## Short summary
This assertion method checks if the current value is inside a limit

**Attention:** 
	limits are included: ``valueIsInRangeOf(ldt#1970-01-01-0:0:0, ldt#1970-01-01-0:0:0, ldt#1970-01-01-0:0:0)``
	is a true assertion

.. <legal notes>

legal notes
=================
| SPDX-FileCopyrightText: © 2022 ekvip automation GmbH <info@ekvip.de>
| SPDX-License-Identifier: Apache-2.0
| For details check: Apache-2.0_

.. _Apache-2.0: https://www.apache.org/licenses/LICENSE-2.0

.. </legal notes>



*)

METHOD valueIsInRangeOf
VAR_INPUT
	(* lower limit for the current value *)
	lowerLimit		:LDT;
	(* current value to check *)
	currentValue	:LDT;
	(* upper limit for the current value *)
	upperLimit		:LDT;
	(* message if the assertion is false *)
	message			:AssertMessage;
END_VAR
IF (
	(currentValue < lowerLimit)
	OR (currentValue > upperLimit)
) THEN
	THIS^.assertionWasWrong(message, THIS^.getDebugInfo('valueIsInRangeOf'));
END_IF
END_METHOD

(*

## Short summary
This assertion method checks if the current value is less than the greater value

.. <legal notes>

legal notes
=================
| SPDX-FileCopyrightText: © 2022 ekvip automation GmbH <info@ekvip.de>
| SPDX-License-Identifier: Apache-2.0
| For details check: Apache-2.0_

.. _Apache-2.0: https://www.apache.org/licenses/LICENSE-2.0

.. </legal notes>



*)

METHOD valueIsLessThan
VAR_INPUT
	(* current value to check *)
	currentValue	:LDT;
	(* greater than upper limit *)
	greaterValue	:LDT;
	(* message if the assertion is false *)
	message			:AssertMessage;
END_VAR
IF (currentValue >= greaterValue) THEN
	THIS^.assertionWasWrong(message, THIS^.getDebugInfo('valueIsLessThan'));
END_IF
END_METHOD

(*

## Short summary
This assertion method checks if the current value is less than or equal to the maximum value

.. <legal notes>

legal notes
=================
| SPDX-FileCopyrightText: © 2022 ekvip automation GmbH <info@ekvip.de>
| SPDX-License-Identifier: Apache-2.0
| For details check: Apache-2.0_

.. _Apache-2.0: https://www.apache.org/licenses/LICENSE-2.0

.. </legal notes>



*)

METHOD valueIsMax
VAR_INPUT
	(* current value to check *)
	currentValue	:LDT;
	(* upper limit for the current value *)
	maximumValue	:LDT;
	(* message if the assertion is false *)
	message			:AssertMessage;
END_VAR
IF (currentValue > maximumValue) THEN
	THIS^.assertionWasWrong(message, THIS^.getDebugInfo('valueIsMax'));
END_IF
END_METHOD

(*

## Short summary
This assertion method checks if the current value is greater than or equal to the minimum value

.. <legal notes>

legal notes
=================
| SPDX-FileCopyrightText: © 2022 ekvip automation GmbH <info@ekvip.de>
| SPDX-License-Identifier: Apache-2.0
| For details check: Apache-2.0_

.. _Apache-2.0: https://www.apache.org/licenses/LICENSE-2.0

.. </legal notes>



*)

METHOD valueIsMin
VAR_INPUT
	(* current value to check *)
	currentValue	:LDT;
	(* lower limit for the current value *)
	minimumValue	:LDT;
	(* message if the assertion is false *)
	message			:AssertMessage;
END_VAR
IF (currentValue < minimumValue) THEN
	THIS^.assertionWasWrong(message, THIS^.getDebugInfo('valueIsMin'));
END_IF
END_METHOD

(*

## Short summary
This assertion method checks if the current value is not equal to the unexpected value

.. <legal notes>

legal notes
=================
| SPDX-FileCopyrightText: © 2022 ekvip automation GmbH <info@ekvip.de>
| SPDX-License-Identifier: Apache-2.0
| For details check: Apache-2.0_

.. _Apache-2.0: https://www.apache.org/licenses/LICENSE-2.0

.. </legal notes>



*)

METHOD valueIsNotEqualTo
VAR_INPUT
	(* current value to check *)
	currentValue	:LDT;
	(* unexpected value to compare *)
	unexpectedValue	:LDT;
	(* message if the assertion is false *)
	message			:AssertMessage;
END_VAR
IF (currentValue = unexpectedValue) THEN
	THIS^.assertionWasWrong(message, THIS^.getDebugInfo('valueIsNotEqualTo'));
END_IF
END_METHOD

END_FUNCTION_BLOCK

// ---- Assertor/Assertions/DateAndTimeAssertions/64Bit/LTOD/classes/TimeOfDayAssertions64Bit.TcPOU
(*

## Short summary
This class provides assert statements for 32 bit time of day ``LTOD``.

.. <legal notes>

legal notes
=================
| SPDX-FileCopyrightText: © 2022 ekvip automation GmbH <info@ekvip.de>
| SPDX-License-Identifier: Apache-2.0
| For details check: Apache-2.0_

.. _Apache-2.0: https://www.apache.org/licenses/LICENSE-2.0

.. </legal notes>



*)

{attribute 'reflection'}
FUNCTION_BLOCK INTERNAL TimeOfDayAssertions64Bit EXTENDS AbstractAssertion IMPLEMENTS I64BitTodAssertions
VAR
END_VAR

(*

## Short summary
This abstract property returns the class name of the concrete object, 
It's for debugging purpose

.. <legal notes>

legal notes
=================
| SPDX-FileCopyrightText: © 2022 ekvip automation GmbH <info@ekvip.de>
| SPDX-License-Identifier: Apache-2.0
| For details check: Apache-2.0_

.. _Apache-2.0: https://www.apache.org/licenses/LICENSE-2.0

.. </legal notes>

*)

PROPERTY className :CNM_AbstractObject.ClassName
GET
className := 'CNM_Assertor.TimeOfDayAssertions64Bit';
END_GET
END_PROPERTY

(*

## Short summary
This assertion method checks if the current value is equal to the expected value

.. <legal notes>

legal notes
=================
| SPDX-FileCopyrightText: © 2022 ekvip automation GmbH <info@ekvip.de>
| SPDX-License-Identifier: Apache-2.0
| For details check: Apache-2.0_

.. _Apache-2.0: https://www.apache.org/licenses/LICENSE-2.0

.. </legal notes>



*)

METHOD valueIsEqualTo
VAR_INPUT
	(* current value to check *)
	currentValue	:LTOD;
	(* expected value to compare *)
	expectedValue	:LTOD;
	(* message if the assertion is false *)
	message			:AssertMessage;
END_VAR
IF (currentValue <> expectedValue) THEN
	THIS^.assertionWasWrong(message, THIS^.getDebugInfo('valueIsEqualTo'));
END_IF
END_METHOD

(*

## Short summary
This assertion method checks if the current value is greater than the less value

.. <legal notes>

legal notes
=================
| SPDX-FileCopyrightText: © 2022 ekvip automation GmbH <info@ekvip.de>
| SPDX-License-Identifier: Apache-2.0
| For details check: Apache-2.0_

.. _Apache-2.0: https://www.apache.org/licenses/LICENSE-2.0

.. </legal notes>



*)

METHOD valueIsGreaterThan
VAR_INPUT
	(* current value to check *)
	currentValue	:LTOD;
	(* less than lower limit *)
	lessValue		:LTOD;
	(* message if the assertion is false *)
	message			:AssertMessage;
END_VAR
IF (currentValue <= lessValue) THEN
	THIS^.assertionWasWrong(message, THIS^.getDebugInfo('valueIsGreaterThan'));
END_IF
END_METHOD

(*

## Short summary
This assertion method checks if the current value is inside a limit

**Attention:** 
	limits are included: ``valueIsInRangeOf(ltod#3:0:0, ltod#3:0:0, ltod#3:0:0)`` is a true assertion

.. <legal notes>

legal notes
=================
| SPDX-FileCopyrightText: © 2022 ekvip automation GmbH <info@ekvip.de>
| SPDX-License-Identifier: Apache-2.0
| For details check: Apache-2.0_

.. _Apache-2.0: https://www.apache.org/licenses/LICENSE-2.0

.. </legal notes>



*)

METHOD valueIsInRangeOf
VAR_INPUT
	(* lower limit for the current value *)
	lowerLimit		:LTOD;
	(* current value to check *)
	currentValue	:LTOD;
	(* upper limit for the current value *)
	upperLimit		:LTOD;
	(* message if the assertion is false *)
	message			:AssertMessage;
END_VAR
IF (
	(currentValue < lowerLimit)
	OR (currentValue > upperLimit)
) THEN
	THIS^.assertionWasWrong(message, THIS^.getDebugInfo('valueIsInRangeOf'));
END_IF
END_METHOD

(*

## Short summary
This assertion method checks if the current value is less than the greater value

.. <legal notes>

legal notes
=================
| SPDX-FileCopyrightText: © 2022 ekvip automation GmbH <info@ekvip.de>
| SPDX-License-Identifier: Apache-2.0
| For details check: Apache-2.0_

.. _Apache-2.0: https://www.apache.org/licenses/LICENSE-2.0

.. </legal notes>



*)

METHOD valueIsLessThan
VAR_INPUT
	(* current value to check *)
	currentValue	:LTOD;
	(* greater than upper limit *)
	greaterValue	:LTOD;
	(* message if the assertion is false *)
	message			:AssertMessage;
END_VAR
IF (currentValue >= greaterValue) THEN
	THIS^.assertionWasWrong(message, THIS^.getDebugInfo('valueIsLessThan'));
END_IF
END_METHOD

(*

## Short summary
This assertion method checks if the current value is less than or equal to the maximum value

.. <legal notes>

legal notes
=================
| SPDX-FileCopyrightText: © 2022 ekvip automation GmbH <info@ekvip.de>
| SPDX-License-Identifier: Apache-2.0
| For details check: Apache-2.0_

.. _Apache-2.0: https://www.apache.org/licenses/LICENSE-2.0

.. </legal notes>



*)

METHOD valueIsMax
VAR_INPUT
	(* current value to check *)
	currentValue	:LTOD;
	(* upper limit for the current value *)
	maximumValue	:LTOD;
	(* message if the assertion is false *)
	message			:AssertMessage;
END_VAR
IF (currentValue > maximumValue) THEN
	THIS^.assertionWasWrong(message, THIS^.getDebugInfo('valueIsMax'));
END_IF
END_METHOD

(*

## Short summary
This assertion method checks if the current value is greater than or equal to the minimum value

.. <legal notes>

legal notes
=================
| SPDX-FileCopyrightText: © 2022 ekvip automation GmbH <info@ekvip.de>
| SPDX-License-Identifier: Apache-2.0
| For details check: Apache-2.0_

.. _Apache-2.0: https://www.apache.org/licenses/LICENSE-2.0

.. </legal notes>



*)

METHOD valueIsMin
VAR_INPUT
	(* current value to check *)
	currentValue	:LTOD;
	(* lower limit for the current value *)
	minimumValue	:LTOD;
	(* message if the assertion is false *)
	message			:AssertMessage;
END_VAR
IF (currentValue < minimumValue) THEN
	THIS^.assertionWasWrong(message, THIS^.getDebugInfo('valueIsMin'));
END_IF
END_METHOD

(*

## Short summary
This assertion method checks if the current value is not equal to the unexpected value

.. <legal notes>

legal notes
=================
| SPDX-FileCopyrightText: © 2022 ekvip automation GmbH <info@ekvip.de>
| SPDX-License-Identifier: Apache-2.0
| For details check: Apache-2.0_

.. _Apache-2.0: https://www.apache.org/licenses/LICENSE-2.0

.. </legal notes>



*)

METHOD valueIsNotEqualTo
VAR_INPUT
	(* current value to check *)
	currentValue	:LTOD;
	(* unexpected value to compare *)
	unexpectedValue	:LTOD;
	(* message if the assertion is false *)
	message			:AssertMessage;
END_VAR
IF (currentValue = unexpectedValue) THEN
	THIS^.assertionWasWrong(message, THIS^.getDebugInfo('valueIsNotEqualTo'));
END_IF
END_METHOD

END_FUNCTION_BLOCK

// ---- Assertor/Assertions/FloatAssertions/classes/FloatAssertions.TcPOU
(*

## Short summary

This class provides assert statements for floatings (``REAL`` and ``LREAL``)
For 32 bit floats (``REAL``) use `FloatAssertions.single`
For 64 bit floats (``LREAL``) use `FloatAssertions.double`

.. <legal notes>

legal notes
=================
| SPDX-FileCopyrightText: © 2022 ekvip automation GmbH <info@ekvip.de>
| SPDX-License-Identifier: Apache-2.0
| For details check: Apache-2.0_

.. _Apache-2.0: https://www.apache.org/licenses/LICENSE-2.0

.. </legal notes>



*)

{attribute 'reflection'}
FUNCTION_BLOCK INTERNAL FloatAssertions EXTENDS CNM_AbstractObject.Object IMPLEMENTS IFloatAssertions, IAssertCallBacksetter
VAR
	(* class to handle assert statements for 32 bit floats *)
	realAssertions	:RealAssertions();
	(* class to handle assert statements for 64 bit floats *)
	lRealAssertions	:LrealAssertions();
END_VAR

(*

## Short summary
This abstract property returns the class name of the concrete object, 
It's for debugging purpose

.. <legal notes>

legal notes
=================
| SPDX-FileCopyrightText: © 2022 ekvip automation GmbH <info@ekvip.de>
| SPDX-License-Identifier: Apache-2.0
| For details check: Apache-2.0_

.. _Apache-2.0: https://www.apache.org/licenses/LICENSE-2.0

.. </legal notes>

*)

PROPERTY className :CNM_AbstractObject.ClassName
GET
className := 'CNM_Assertor.FloatAssertions';
END_GET
END_PROPERTY

(*

## Short summary
Returns the interface `ILrealAssertions` with assert statements for 64 bit floatings (``LREAL``)

.. <legal notes>

legal notes
=================
| SPDX-FileCopyrightText: © 2022 ekvip automation GmbH <info@ekvip.de>
| SPDX-License-Identifier: Apache-2.0
| For details check: Apache-2.0_

.. _Apache-2.0: https://www.apache.org/licenses/LICENSE-2.0

.. </legal notes>

*)

PROPERTY double :ILrealAssertions
GET
double := THIS^.lRealAssertions;
END_GET
END_PROPERTY

(*

## Short summary
This methods is the setter for the callback class if an assertion was false

.. <legal notes>

legal notes
=================
| SPDX-FileCopyrightText: © 2022 ekvip automation GmbH <info@ekvip.de>
| SPDX-License-Identifier: Apache-2.0
| For details check: Apache-2.0_

.. _Apache-2.0: https://www.apache.org/licenses/LICENSE-2.0

.. </legal notes>



*)

METHOD setCallBack
VAR_INPUT
	(* the class that must be informed if an assertion is false *)
	callBack	:IAssertCallBack;  
END_VAR
THIS^.realAssertions.setCallBack(callBack);
THIS^.lRealAssertions.setCallBack(callBack);
END_METHOD

(*

## Short summary
Returns the interface `IRealAssertions` with assert statements for 32 bit floatings (``REAL``)

.. <legal notes>

legal notes
=================
| SPDX-FileCopyrightText: © 2022 ekvip automation GmbH <info@ekvip.de>
| SPDX-License-Identifier: Apache-2.0
| For details check: Apache-2.0_

.. _Apache-2.0: https://www.apache.org/licenses/LICENSE-2.0

.. </legal notes>

*)

PROPERTY single :IRealAssertions
GET
single := THIS^.realAssertions;
END_GET
END_PROPERTY

END_FUNCTION_BLOCK

// ---- Assertor/Assertions/FloatAssertions/Real/classes/RealAssertions.TcPOU
(*

## Short summary
This class provides assert statements for 32 bit floatings (``REAL``).
It implements the interface `IRealAssertions`

.. <legal notes>

legal notes
=================
| SPDX-FileCopyrightText: © 2022 ekvip automation GmbH <info@ekvip.de>
| SPDX-License-Identifier: Apache-2.0
| For details check: Apache-2.0_

.. _Apache-2.0: https://www.apache.org/licenses/LICENSE-2.0

.. </legal notes>



*)

{attribute 'reflection'}
FUNCTION_BLOCK INTERNAL RealAssertions EXTENDS AbstractAssertion IMPLEMENTS IRealAssertions
VAR
END_VAR
VAR CONSTANT
	(* mask for determining value as a special value *)
	MASK_FOR_EXPONENT 	:DWORD := 16#7F80_0000;
	(* mask for determining a special value as NaN or infinite *)  
	MASK_FOR_FRACTION	:DWORD := 16#007F_FFFF;
	(* mask to get the sign bit of an infinite or zero value *)
	MASK_FOR_SIGN_BIT	:DWORD := 16#8000_0000;
	(* just to compare results or the memory of a float value *)
	ZERO				:DWORD := 16#0000_0000;
END_VAR

(*

## Short summary
This abstract property returns the class name of the concrete object, 
It's for debugging purpose

.. <legal notes>

legal notes
=================
| SPDX-FileCopyrightText: © 2022 ekvip automation GmbH <info@ekvip.de>
| SPDX-License-Identifier: Apache-2.0
| For details check: Apache-2.0_

.. _Apache-2.0: https://www.apache.org/licenses/LICENSE-2.0

.. </legal notes>

*)

PROPERTY className :CNM_AbstractObject.ClassName
GET
className := 'CNM_Assertor.RealAssertions';
END_GET
END_PROPERTY

(*

## Short summary
This method checks if a value is infinite
(infinity OR -inifinity), for details check [IEEE 754](https://en.wikipedia.org/wiki/IEEE_754)


.. <legal notes>

legal notes
=================
| SPDX-FileCopyrightText: © 2023 ekvip automation GmbH <info@ekvip.de>
| SPDX-License-Identifier: Apache-2.0
| For details check: Apache-2.0_

.. _Apache-2.0: https://www.apache.org/licenses/LICENSE-2.0

.. </legal notes>


:return: 
``TRUE``: value is inifinty or -infinity
``FALSE``: value is not inifinty and not -infinity

*)

METHOD PROTECTED isValueInfinite :BOOL
VAR_INPUT
	(* value to check *)
	value			:REAL;	
END_VAR
VAR
	(* just to cast the value*)
	realAsDword	:POINTER TO DWORD;
END_VAR
realAsDword := ADR(value);
isValueInfinite := (
	THIS^.isValueSpecial(value)
	AND_THEN ((realAsDword^ AND THIS^.MASK_FOR_FRACTION) = THIS^.ZERO)
);
END_METHOD

(*

## Short summary
This method checks if a value is not a number
(NaN), for details check [IEEE 754](https://en.wikipedia.org/wiki/IEEE_754)


.. <legal notes>

legal notes
=================
| SPDX-FileCopyrightText: © 2023 ekvip automation GmbH <info@ekvip.de>
| SPDX-License-Identifier: Apache-2.0
| For details check: Apache-2.0_

.. _Apache-2.0: https://www.apache.org/licenses/LICENSE-2.0

.. </legal notes>


:return: 
``TRUE``: value is NaN
``FALSE``: value is not NaN

*)

METHOD PROTECTED isValueNaN :BOOL
VAR_INPUT
	(* value to check *)
	value			:REAL;	
END_VAR
VAR
	(* just to cast the value*)
	realAsDword	:POINTER TO DWORD;
END_VAR
realAsDword := ADR(value);
isValueNaN := (
	THIS^.isValueSpecial(value)
	AND_THEN ((realAsDword^ AND THIS^.MASK_FOR_FRACTION) > THIS^.ZERO)
);
END_METHOD

(*

## Short summary
This method checks if a value is negative infinite
(-inifinity), for details check [IEEE 754](https://en.wikipedia.org/wiki/IEEE_754)


.. <legal notes>

legal notes
=================
| SPDX-FileCopyrightText: © 2023 ekvip automation GmbH <info@ekvip.de>
| SPDX-License-Identifier: Apache-2.0
| For details check: Apache-2.0_

.. _Apache-2.0: https://www.apache.org/licenses/LICENSE-2.0

.. </legal notes>


:return: 
``TRUE``: value is -infinity
``FALSE``: value is not -infinity

*)

METHOD PROTECTED isValueNegativeInfinite : BOOL
VAR_INPUT
	(* value to check *)
	value			:REAL;	
END_VAR
VAR
	(* just to cast the value*)
	realAsDword	:POINTER TO DWORD;
END_VAR
realAsDword := ADR(value);
isValueNegativeInfinite := (
	THIS^.isValueInfinite(value)
	AND_THEN ((realAsDword^ AND THIS^.MASK_FOR_SIGN_BIT) = THIS^.MASK_FOR_SIGN_BIT)
);
END_METHOD

(*

## Short summary
This method checks if a value is positive infinite
(infinity), for details check [IEEE 754](https://en.wikipedia.org/wiki/IEEE_754)


.. <legal notes>

legal notes
=================
| SPDX-FileCopyrightText: © 2023 ekvip automation GmbH <info@ekvip.de>
| SPDX-License-Identifier: Apache-2.0
| For details check: Apache-2.0_

.. _Apache-2.0: https://www.apache.org/licenses/LICENSE-2.0

.. </legal notes>


:return: 
``TRUE``: value is inifinty
``FALSE``: value is not inifinty

*)

METHOD PROTECTED isValuePositiveInfinite :BOOL
VAR_INPUT
	(* value to check *)
	value			:REAL;	
END_VAR
VAR
	(* just to cast the value*)
	realAsDword	:POINTER TO DWORD;
END_VAR
realAsDword := ADR(value);
isValuePositiveInfinite := (
	THIS^.isValueInfinite(value)
	AND_THEN ((realAsDword^ AND THIS^.MASK_FOR_SIGN_BIT) = THIS^.ZERO)
);
END_METHOD

(*

## Short summary
This method checks if a value is a special value
(NaN OR infinity OR -inifinity), for details check [IEEE 754](https://en.wikipedia.org/wiki/IEEE_754)


.. <legal notes>

legal notes
=================
| SPDX-FileCopyrightText: © 2023 ekvip automation GmbH <info@ekvip.de>
| SPDX-License-Identifier: Apache-2.0
| For details check: Apache-2.0_

.. _Apache-2.0: https://www.apache.org/licenses/LICENSE-2.0

.. </legal notes>


:return: 
``TRUE``: value is inifinty or -infinity or NaN
``FALSE``: value is not inifinty and not -infinity and not NaN

*)

METHOD PROTECTED isValueSpecial :BOOL
VAR_INPUT
	(* value to check *)
	value			:REAL;	
END_VAR
VAR
	(* just to cast the value*)
	realAsDword	:POINTER TO DWORD;
END_VAR
realAsDword := ADR(value);
isValueSpecial := ((realAsDword^ AND THIS^.MASK_FOR_EXPONENT) = THIS^.MASK_FOR_EXPONENT);
END_METHOD

(*

## Short summary
This assertion method checks if the current value is a number (NOT NaN)
for details check [IEEE 754](https://en.wikipedia.org/wiki/IEEE_754)


.. <legal notes>

legal notes
=================
| SPDX-FileCopyrightText: © 2023 ekvip automation GmbH <info@ekvip.de>
| SPDX-License-Identifier: Apache-2.0
| For details check: Apache-2.0_

.. _Apache-2.0: https://www.apache.org/licenses/LICENSE-2.0

.. </legal notes>



*)

METHOD valueIsANumber
VAR_INPUT
	(* current value to check *)
	currentValue	:REAL;
	(* message if the assertion is false *)
	message			:AssertMessage;
END_VAR
IF (THIS^.isValueNaN(currentValue)) THEN
	THIS^.assertionWasWrong(message, THIS^.getDebugInfo('valueIsANumber'));
END_IF
END_METHOD

(*

## Short summary
This assertion method checks if the current value is equal to the expected value

**Attention:** 
	Nothing is equal to NaN, that means if ``currentValue`` OR ``expectedValue`` OR ``tolerance``
	is NaN then is the assertion false. For details check `IEEE 754`_

**Attention:** 
	infinity is equal to infinity and -infinity is equal to -infinity, that means if
	``currentValue`` AND ``expectedValue`` have the value infinity 
	OR ``currentValue`` AND ``expectedValue`` have the value -infinity
	the assertion is TRUE. For details check `IEEE 754`_

**Attention:** 
	If ``tolerance`` has the value infinity or -infinity and 
	``currentValue`` is not NaN and ``expectedValue`` is not NaN
	then is the assertion true. for details check [IEEE 754](https://en.wikipedia.org/wiki/IEEE_754)


.. <legal notes>

legal notes
=================
| SPDX-FileCopyrightText: © 2022 ekvip automation GmbH <info@ekvip.de>
| SPDX-License-Identifier: Apache-2.0
| For details check: Apache-2.0_

.. _Apache-2.0: https://www.apache.org/licenses/LICENSE-2.0

.. </legal notes>



*)

METHOD valueIsEqualTo
VAR_INPUT
	(* current value to check *)
	currentValue	:REAL;
	(* expected value to compare *)
	expectedValue	:REAL;
	(* tolerance to compensate twiddling floats, it has no sign *)
	tolerance		:REAL;
	(* message if the assertion is false *)
	message			:AssertMessage;
END_VAR
IF (
	THIS^.isValueNaN(currentValue)
	OR_ELSE THIS^.isValueNaN(expectedValue)
	OR_ELSE THIS^.isValueNaN(tolerance)
) THEN
	THIS^.assertionWasWrong(message, THIS^.getDebugInfo('valueIsEqualTo'));
ELSIF (THIS^.isValueInfinite(tolerance)) THEN
	RETURN;
ELSIF (
	THIS^.isValueInfinite(currentValue)
	OR_ELSE THIS^.isValueInfinite(expectedValue)
	OR_ELSE THIS^.isValueInfinite(tolerance)
) THEN
	RETURN (THIS^.isValuePositiveInfinite(currentValue) AND_THEN THIS^.isValuePositiveInfinite(expectedValue));
	RETURN (THIS^.isValueNegativeInfinite(currentValue) AND_THEN THIS^.isValueNegativeInfinite(expectedValue));
	THIS^.assertionWasWrong(message, THIS^.getDebugInfo('valueIsEqualTo'));	
ELSIF (ABS(currentValue-expectedValue) > ABS(tolerance)) THEN
	THIS^.assertionWasWrong(message, THIS^.getDebugInfo('valueIsEqualTo'));
END_IF
END_METHOD

(*

## Short summary
This assertion method checks if the current value is finite
(NOT (infinity OR -inifinity)), for details check [IEEE 754](https://en.wikipedia.org/wiki/IEEE_754)


.. <legal notes>

legal notes
=================
| SPDX-FileCopyrightText: © 2023 ekvip automation GmbH <info@ekvip.de>
| SPDX-License-Identifier: Apache-2.0
| For details check: Apache-2.0_

.. _Apache-2.0: https://www.apache.org/licenses/LICENSE-2.0

.. </legal notes>



*)

METHOD valueIsFinite
VAR_INPUT
	(* current value to check *)
	currentValue	:REAL;
	(* message if the assertion is false *)
	message			:AssertMessage;
END_VAR
IF (THIS^.isValueInfinite(currentValue)) THEN
	THIS^.assertionWasWrong(message, THIS^.getDebugInfo('valueIsFinite'));
END_IF
END_METHOD

(*

## Short summary
This assertion method checks if the current value is greater than the less value

**Attention:** 
	Any comparsion to NaN is ``FALSE`` that means if ``currentValue`` OR ``lessValue``
	is NaN then is the assertion false.
	For details check `IEEE 754`_ and the truth table below.

**Attention:** 
	Every number is smaller than infinity except infinity, it's equal.
	Every number is greater than -infinity except -infinity, it's equal.
	For details check [IEEE 754](https://en.wikipedia.org/wiki/IEEE_754) and the truth table below.


truth table for special values
===============================
+----------------------+-------------------+---------------+
| **``currentValue``** | **``lessValue``** | **assertion** |
+======================+===================+===============+
| NaN                  | Any value         | FASLE         |
+----------------------+-------------------+---------------+
| Any value            | NaN               | FALSE         |
+----------------------+-------------------+---------------+
| infinity             | NOT NaN           | TRUE          |
|                      | NOT infinity      |               |
+----------------------+-------------------+---------------+
| -infinity             | Any value         | FALSE         |
+----------------------+-------------------+---------------+
| Any value            | infinity          | FALSE         |
+----------------------+-------------------+---------------+
| NOT NaN              | -inifinity        | TRUE          |
| NOT -infinity        |                   |               |
+----------------------+-------------------+---------------+

.. <legal notes>

legal notes
=================
| SPDX-FileCopyrightText: © 2022 ekvip automation GmbH <info@ekvip.de>
| SPDX-License-Identifier: Apache-2.0
| For details check: Apache-2.0_

.. _Apache-2.0: https://www.apache.org/licenses/LICENSE-2.0

.. </legal notes>



*)

METHOD valueIsGreaterThan
VAR_INPUT
	(* current value to check *)
	currentValue	:REAL;
	(* less than lower limit *)
	lessValue		:REAL;
	(* message if the assertion is false *)
	message			:AssertMessage;
END_VAR
IF (
	THIS^.isValueNaN(currentValue) 
	OR_ELSE THIS^.isValueNaN(lessValue)
	OR_ELSE THIS^.isValueNegativeInfinite(currentValue) 
	OR_ELSE THIS^.isValuePositiveInfinite(lessValue)
)THEN
	THIS^.assertionWasWrong(message, THIS^.getDebugInfo('valueIsGreaterThan'));
ELSIF (
	THIS^.isValueNegativeInfinite(lessValue)
	OR_ELSE THIS^.isValuePositiveInfinite(currentValue)
) THEN
	RETURN;
ELSIF (currentValue <= lessValue) THEN
	THIS^.assertionWasWrong(message, THIS^.getDebugInfo('valueIsGreaterThan'));
END_IF
END_METHOD

(*

## Short summary
This assertion method checks if the current value is infinite
(infinity OR -inifinity), for details check [IEEE 754](https://en.wikipedia.org/wiki/IEEE_754)


.. <legal notes>

legal notes
=================
| SPDX-FileCopyrightText: © 2023 ekvip automation GmbH <info@ekvip.de>
| SPDX-License-Identifier: Apache-2.0
| For details check: Apache-2.0_

.. _Apache-2.0: https://www.apache.org/licenses/LICENSE-2.0

.. </legal notes>



*)

METHOD valueIsInfinite
VAR_INPUT
	(* current value to check *)
	currentValue	:REAL;
	(* message if the assertion is false *)
	message			:AssertMessage;
END_VAR
IF (NOT THIS^.isValueInfinite(currentValue)) THEN
	THIS^.assertionWasWrong(message, THIS^.getDebugInfo('valueIsInfinite'));
END_IF
END_METHOD

(*

## Short summary
This assertion method checks if the current value is inside a limit

**Attention:** 
	limits are included: ``valueIsInRangeOf(3.0, 3.0, 3.0)`` is a true assertion

**Attention:** 
	Any comparsion to NaN is ``FALSE`` that means 
	if ``lowerLimit`` OR ``currentValue`` OR ``upperLimit``
	is NaN then is the assertion false.
	For details check `IEEE 754`_ and the truth table below.

**Attention:** 
	Every number is smaller than infinity except infinity, it's equal.
	Every number is greater than -infinity except -infinity, it's equal.
	For details check [IEEE 754](https://en.wikipedia.org/wiki/IEEE_754) and the truth table below.


truth table for special values
===============================
+--------------------+----------------------+--------------------+---------------+
| **``lowerLimit``** | **``currentValue``** | **``upperLimit``** | **assertion** |
+====================+======================+====================+===============+
| NaN                | Any value            | Any value          | FASLE         |
+--------------------+----------------------+--------------------+---------------+
| Any value          | NaN                  | Any value          | FALSE         |
+--------------------+----------------------+--------------------+---------------+
| Any value          | Any value            | NaN                | FALSE         |
+--------------------+----------------------+--------------------+---------------+
| -infinity          | NOT NaN              | infinity           | TRUE          |
+--------------------+----------------------+--------------------+---------------+
| infinity           | Any value            | -infinity          | FALSE         |
+--------------------+----------------------+--------------------+---------------+
| NOT -infinity      | -infinity            | Any value          | FALSE         |
+--------------------+----------------------+--------------------+---------------+
| Any value          | infinity             | NOT infinity       | FALSE         |
+--------------------+----------------------+--------------------+---------------+
| -infinity          | -infinity            | -infinity          | TRUE          |
+--------------------+----------------------+--------------------+---------------+
| infinity           | infinity             | infinity           | TRUE          |
+--------------------+----------------------+--------------------+---------------+
| -infinity          | NOT -infinity        | -infinity          | FALSE         |
+--------------------+----------------------+--------------------+---------------+
| infinity           | NOT infinity         | infinity           | FALSE         |
+--------------------+----------------------+--------------------+---------------+

.. <legal notes>

legal notes
=================
| SPDX-FileCopyrightText: © 2022 ekvip automation GmbH <info@ekvip.de>
| SPDX-License-Identifier: Apache-2.0
| For details check: Apache-2.0_

.. _Apache-2.0: https://www.apache.org/licenses/LICENSE-2.0

.. </legal notes>



*)

METHOD valueIsInRangeOf
VAR_INPUT
	(* lower limit for the current value *)
	lowerLimit		:REAL;
	(* current value to check *)
	currentValue	:REAL;
	(* upper limit for the current value *)
	upperLimit		:REAL;
	(* message if the assertion is false *)
	message			:AssertMessage;
END_VAR
IF (
	THIS^.isValueNaN(lowerLimit)
	OR_ELSE THIS^.isValueNaN(currentValue)
	OR_ELSE THIS^.isValueNaN(upperLimit)
	OR_ELSE (
		THIS^.isValueNegativeInfinite(upperLimit) 
		AND_THEN THIS^.isValuePositiveInfinite(lowerLimit)
	) OR_ELSE (	
		THIS^.isValueNegativeInfinite(currentValue) 
		AND_THEN (NOT THIS^.isValueNegativeInfinite(lowerLimit))
	) OR_ELSE (
		THIS^.isValuePositiveInfinite(currentValue) 
		AND_THEN (NOT THIS^.isValuePositiveInfinite(upperLimit))
	) OR_ELSE (
		THIS^.isValuePositiveInfinite(lowerLimit)
		AND_THEN (NOT THIS^.isValuePositiveInfinite(currentValue))
		AND_THEN THIS^.isValuePositiveInfinite(upperLimit)
	) OR_ELSE (
		THIS^.isValueNegativeInfinite(lowerLimit)
		AND_THEN (NOT THIS^.isValueNegativeInfinite(currentValue))
		AND_THEN THIS^.isValueNegativeInfinite(upperLimit))
) THEN
	THIS^.assertionWasWrong(message, THIS^.getDebugInfo('valueIsInRangeOf'));
ELSIF ((
		THIS^.isValuePositiveInfinite(lowerLimit)
		AND_THEN THIS^.isValuePositiveInfinite(currentValue)
		AND_THEN THIS^.isValuePositiveInfinite(upperLimit)
	) OR_ELSE (
		THIS^.isValueNegativeInfinite(lowerLimit)
		AND_THEN THIS^.isValueNegativeInfinite(currentValue)
		AND_THEN THIS^.isValueNegativeInfinite(upperLimit)
	) OR_ELSE (
		THIS^.isValueNegativeInfinite(lowerLimit) 
		AND_THEN THIS^.isValuePositiveInfinite(upperLimit))
) THEN
	RETURN;
ELSIF ((currentValue < lowerLimit) OR (currentValue > upperLimit)) THEN
	THIS^.assertionWasWrong(message, THIS^.getDebugInfo('valueIsInRangeOf'));
END_IF
END_METHOD

(*

## Short summary
This assertion method checks if the current value is greater than the less value

**Attention:**
	Any comparsion to NaN is ``FALSE`` that means if ``currentValue`` OR ``greaterValue``
	is NaN then is the assertion false.
	For details check `IEEE 754`_ and the truth table below.

**Attention:**
	Every number is smaller than infinity except infinity, it's equal.
	Every number is greater than -infinity except -infinity, it's equal.
	For details check [IEEE 754](https://en.wikipedia.org/wiki/IEEE_754) and the truth table below.


truth table for special values
===============================
+----------------------+----------------------+---------------+
| **``currentValue``** | **``greaterValue``** | **assertion** |
+======================+======================+===============+
| NaN                  | Any value            | FASLE         |
+----------------------+----------------------+---------------+
| Any value            | NaN                  | FALSE         |
+----------------------+----------------------+---------------+
| infinity             | Any value            | FALSE         |
+----------------------+----------------------+---------------+
| -infinity             | NOT NaN              | TRUE          |
|                      | NOT -infinity        |               |
+----------------------+----------------------+---------------+
| NOT NaN              | infinity             | TRUE          |
| NOT infinity         |                      |               |
+----------------------+----------------------+---------------+

.. <legal notes>

legal notes
=================
| SPDX-FileCopyrightText: © 2022 ekvip automation GmbH <info@ekvip.de>
| SPDX-License-Identifier: Apache-2.0
| For details check: Apache-2.0_

.. _Apache-2.0: https://www.apache.org/licenses/LICENSE-2.0

.. </legal notes>



*)

METHOD valueIsLessThan
VAR_INPUT
	(* current value to check *)
	currentValue	:REAL;
	(* greater than upper limit *)
	greaterValue	:REAL;
	(* message if the assertion is false *)
	message			:AssertMessage;
END_VAR
IF (
	THIS^.isValueNaN(currentValue) 
	OR_ELSE THIS^.isValueNaN(greaterValue)
	OR_ELSE THIS^.isValuePositiveInfinite(currentValue)
	OR_ELSE THIS^.isValueNegativeInfinite(greaterValue)
) THEN
	THIS^.assertionWasWrong(message, THIS^.getDebugInfo('valueIsLessThan'));
ELSIF (
	THIS^.isValuePositiveInfinite(greaterValue)
	OR_ELSE THIS^.isValueNegativeInfinite(currentValue)
) THEN
	RETURN;
ELSIF (currentValue >= greaterValue) THEN
	THIS^.assertionWasWrong(message, THIS^.getDebugInfo('valueIsLessThan'));
END_IF
END_METHOD

(*

## Short summary
This assertion method checks if the current value is less than or equal to the maximum value

**Attention:**
	Any comparsion to NaN is ``FALSE`` that means if ``currentValue`` OR ``maximumValue``
	is NaN then is the assertion false.
	For details check `IEEE 754`_ and the truth table below.

**Attention:**
	Every number is smaller than infinity except infinity, it's equal.
	Every number is greater than -infinity except -infinity, it's equal.
	For details check [IEEE 754](https://en.wikipedia.org/wiki/IEEE_754) and the truth table below.


truth table for special values
===============================
+----------------------+----------------------+---------------+
| **``currentValue``** | **``maximumValue``** | **assertion** |
+======================+======================+===============+
| NaN                  | Any value            | FASLE         |
+----------------------+----------------------+---------------+
| Any value            | NaN                  | FALSE         |
+----------------------+----------------------+---------------+
| NOT NaN              | infinity             | TRUE          |
+----------------------+----------------------+---------------+
| -infinity            | NOT NaN              | TRUE          |
+----------------------+----------------------+---------------+
| infinity             | NOT infinity         | FALSE         |
+----------------------+----------------------+---------------+
| NOT -infinity        | -infinity            | FALSE         |
+----------------------+----------------------+---------------+

.. <legal notes>

legal notes
=================
| SPDX-FileCopyrightText: © 2022 ekvip automation GmbH <info@ekvip.de>
| SPDX-License-Identifier: Apache-2.0
| For details check: Apache-2.0_

.. _Apache-2.0: https://www.apache.org/licenses/LICENSE-2.0

.. </legal notes>



*)

METHOD valueIsMax
VAR_INPUT
	(* current value to check *)
	currentValue	:REAL;
	(* upper limit for the current value *)
	maximumValue	:REAL;
	(* message if the assertion is false *)
	message			:AssertMessage;
END_VAR
IF (
	THIS^.isValueNaN(currentValue) 
	OR_ELSE THIS^.isValueNaN(maximumValue)
	OR_ELSE (
		THIS^.isValueNegativeInfinite(maximumValue)
		AND_THEN (NOT THIS^.isValueNegativeInfinite(currentValue))
	) OR_ELSE (
		THIS^.isValuePositiveInfinite(currentValue)
		AND_THEN (NOT THIS^.isValuePositiveInfinite(maximumValue))
	)
) THEN
	THIS^.assertionWasWrong(message, THIS^.getDebugInfo('valueIsMax'));
ELSIF (
	THIS^.isValuePositiveInfinite(maximumValue)
	OR_ELSE THIS^.isValueNegativeInfinite(currentValue)
) THEN
	RETURN;
ELSIF (currentValue > maximumValue) THEN
	THIS^.assertionWasWrong(message, THIS^.getDebugInfo('valueIsMax'));
END_IF
END_METHOD

(*

## Short summary
This assertion method checks if the current value is greater than or equal to the minimum value

**Attention:**
	Any comparsion to NaN is ``FALSE`` that means if ``currentValue`` OR ``minimumValue``
	is NaN then is the assertion false.
	For details check `IEEE 754`_ and the truth table below.

**Attention:**
	Every number is smaller than infinity except infinity, it's equal.
	Every number is greater than -infinity except -infinity, it's equal.
	For details check [IEEE 754](https://en.wikipedia.org/wiki/IEEE_754) and the truth table below.


truth table for special values
===============================
+----------------------+----------------------+---------------+
| **``currentValue``** | **``minimumValue``** | **assertion** |
+======================+======================+===============+
| NaN                  | Any value            | FASLE         |
+----------------------+----------------------+---------------+
| Any value            | NaN                  | FALSE         |
+----------------------+----------------------+---------------+
| infinity             | NOT NaN              | TRUE          |
+----------------------+----------------------+---------------+
| NOT NaN              | -infinity            | TRUE          |
+----------------------+----------------------+---------------+
| -infinity            | NOT -infinity        | FALSE         |
+----------------------+----------------------+---------------+
| NOT infinity         | infinity             | FALSE         |
+----------------------+----------------------+---------------+

.. <legal notes>

legal notes
=================
| SPDX-FileCopyrightText: © 2022 ekvip automation GmbH <info@ekvip.de>
| SPDX-License-Identifier: Apache-2.0
| For details check: Apache-2.0_

.. _Apache-2.0: https://www.apache.org/licenses/LICENSE-2.0

.. </legal notes>



*)

METHOD valueIsMin
VAR_INPUT
	(* current value to check *)
	currentValue	:REAL;
	(* lower limit for the current value *)
	minimumValue	:REAL;
	(* message if the assertion is false *)
	message			:AssertMessage;
END_VAR
IF (
	THIS^.isValueNaN(currentValue) 
	OR_ELSE THIS^.isValueNaN(minimumValue)
	OR_ELSE (
		THIS^.isValueNegativeInfinite(currentValue)
		AND_THEN (NOT THIS^.isValueNegativeInfinite(minimumValue))
	) OR_ELSE (
		THIS^.isValuePositiveInfinite(minimumValue)
		AND_THEN (NOT THIS^.isValuePositiveInfinite(currentValue))
	)
) THEN
	THIS^.assertionWasWrong(message, THIS^.getDebugInfo('valueIsMin'));
ELSIF (
	THIS^.isValuePositiveInfinite(currentValue)
	OR_ELSE THIS^.isValueNegativeInfinite(minimumValue)
) THEN
	RETURN;
ELSIF (currentValue < minimumValue) THEN
	THIS^.assertionWasWrong(message, THIS^.getDebugInfo('valueIsMin'));
END_IF
END_METHOD

(*

## Short summary
This assertion method checks if the current value is a not a number (NaN)
for details check [IEEE 754](https://en.wikipedia.org/wiki/IEEE_754)


.. <legal notes>

legal notes
=================
| SPDX-FileCopyrightText: © 2023 ekvip automation GmbH <info@ekvip.de>
| SPDX-License-Identifier: Apache-2.0
| For details check: Apache-2.0_

.. _Apache-2.0: https://www.apache.org/licenses/LICENSE-2.0

.. </legal notes>



*)

METHOD valueIsNaN
VAR_INPUT
	(* current value to check *)
	currentValue	:REAL;
	(* message if the assertion is false *)
	message			:AssertMessage;
END_VAR
IF (NOT THIS^.isValueNaN(currentValue)) THEN
	THIS^.assertionWasWrong(message, THIS^.getDebugInfo('valueIsNaN'));
END_IF
END_METHOD

(*

## Short summary
This assertion method checks if the current value is negative

**Attention:**
	Any comparsion to NaN is ``FALSE`` that means if ``currentValue``
	is NaN then is the assertion false.
	For details check `IEEE 754`_.

**Attention:**
	``currentValue`` has the value infinity means the assertion is false.
	``currentValue`` has the value -infinity means the assertion is true.
	``currentValue`` has the +0.0 means the assertion is false.
	``currentValue`` has the value -0.0 means the assertion is true.	
		For details check [IEEE 754](https://en.wikipedia.org/wiki/IEEE_754).


.. <legal notes>

legal notes
=================
| SPDX-FileCopyrightText: © 2022 ekvip automation GmbH <info@ekvip.de>
| SPDX-License-Identifier: Apache-2.0
| For details check: Apache-2.0_

.. _Apache-2.0: https://www.apache.org/licenses/LICENSE-2.0

.. </legal notes>



*)

METHOD valueIsNegative
VAR_INPUT
	(* current value to check *)
	currentValue	:REAL;
	(* message if the assertion is false *)
	message			:AssertMessage;
END_VAR
VAR
	(* just to cast ``currentValue`` *)
	currentValueAsDWord	:POINTER TO DWORD;
END_VAR
IF (THIS^.isValueNaN(currentValue)) THEN	
	THIS^.assertionWasWrong(message, THIS^.getDebugInfo('valueIsNegative'));
ELSE
	currentValueAsDWord := ADR(currentValue);
	IF ((currentValueAsDWord^ AND THIS^.MASK_FOR_SIGN_BIT) = THIS^.ZERO) THEN
		THIS^.assertionWasWrong(message, THIS^.getDebugInfo('valueIsNegative'));
	END_IF
END_IF
END_METHOD

(*

## Short summary
This assertion method checks if the current value is negative infinite
(-infinity), for details check [IEEE 754](https://en.wikipedia.org/wiki/IEEE_754)


.. <legal notes>

legal notes
=================
| SPDX-FileCopyrightText: © 2023 ekvip automation GmbH <info@ekvip.de>
| SPDX-License-Identifier: Apache-2.0
| For details check: Apache-2.0_

.. _Apache-2.0: https://www.apache.org/licenses/LICENSE-2.0

.. </legal notes>



*)

METHOD valueIsNegativeInfinite
VAR_INPUT
	(* current value to check *)
	currentValue	:REAL;
	(* message if the assertion is false *)
	message			:AssertMessage;
END_VAR
IF (NOT THIS^.isValueNegativeInfinite(currentValue)) THEN
	THIS^.assertionWasWrong(message, THIS^.getDebugInfo('valueIsNegativeInfinite'));
END_IF
END_METHOD

(*

## Short summary
This assertion method checks if the current value is -0.0
for details check [IEEE 754](https://en.wikipedia.org/wiki/IEEE_754)


.. <legal notes>

legal notes
=================
| SPDX-FileCopyrightText: © 2023 ekvip automation GmbH <info@ekvip.de>
| SPDX-License-Identifier: Apache-2.0
| For details check: Apache-2.0_

.. _Apache-2.0: https://www.apache.org/licenses/LICENSE-2.0

.. </legal notes>



*)

METHOD valueIsNegativeZero
VAR_INPUT
	(* current value to check *)
	currentValue	:REAL;
	(* message if the assertion is false *)
	message			:AssertMessage;
END_VAR
VAR
	(* just to cast ``currentValue`` *)
	currentValueAsDWord	:POINTER TO DWORD;
END_VAR
currentValueAsDWord := ADR(currentValue);
IF (currentValueAsDWord^ <> THIS^.MASK_FOR_SIGN_BIT) THEN
	THIS^.assertionWasWrong(message, THIS^.getDebugInfo('valueIsNegativeZero'));
END_IF
END_METHOD

(*

## Short summary
This assertion method checks if the current value is a normal number
(a finite non-zero/non-subnormal floating-point number)
for details check [IEEE 754](https://en.wikipedia.org/wiki/IEEE_754)


.. <legal notes>

legal notes
=================
| SPDX-FileCopyrightText: © 2023 ekvip automation GmbH <info@ekvip.de>
| SPDX-License-Identifier: Apache-2.0
| For details check: Apache-2.0_

.. _Apache-2.0: https://www.apache.org/licenses/LICENSE-2.0

.. </legal notes>



*)

METHOD valueIsNormal
VAR_INPUT
	(* current value to check *)
	currentValue	:REAL;
	(* message if the assertion is false *)
	message			:AssertMessage;
END_VAR
VAR
	(* just to cast ``currentValue`` *)
	currentValueAsDWord	:POINTER TO DWORD;
END_VAR
IF (THIS^.isValueNaN(currentValue) OR_ELSE THIS^.isValueInfinite(currentValue)) THEN
	THIS^.assertionWasWrong(message, THIS^.getDebugInfo('valueIsNormal'));
ELSE
	currentValueAsDWord := ADR(currentValue);
	IF ((currentValueAsDWord^ AND THIS^.MASK_FOR_EXPONENT) = THIS^.ZERO) THEN
		THIS^.assertionWasWrong(message, THIS^.getDebugInfo('valueIsNormal'));
	END_IF
END_IF
END_METHOD

(*

## Short summary
This assertion method checks if the current value is not equal to the unexpected value

**Attention:** 
	Nothing is equal to NaN, that means if ``currentValue`` OR ``unexpectedValue`` OR ``tolerance``
	is NaN then is the assertion true. For details check `IEEE 754`_

**Attention:** 
	infinity is equal to infinity and -infinity is equal to -infinity, that means if
	``currentValue`` AND ``unexpectedValue`` have the value infinity 
	OR ``currentValue`` AND ``unexpectedValue`` have the value -infinity
	the assertion is false. For details check `IEEE 754`_

**Attention:** 
	If ``tolerance`` has the value infinity or -infinity and 
	``currentValue`` is not NaN and ``unexpectedValue`` is not NaN
	then is the assertion false. for details check [IEEE 754](https://en.wikipedia.org/wiki/IEEE_754)


.. <legal notes>

legal notes
=================
| SPDX-FileCopyrightText: © 2022 ekvip automation GmbH <info@ekvip.de>
| SPDX-License-Identifier: Apache-2.0
| For details check: Apache-2.0_

.. _Apache-2.0: https://www.apache.org/licenses/LICENSE-2.0

.. </legal notes>



*)

METHOD valueIsNotEqualTo
VAR_INPUT
	(* current value to check *)
	currentValue	:REAL;
	(* unexpected value to compare *)
	unexpectedValue	:REAL;
	(* tolerance to compensate twiddling floats, it has no sign *)
	tolerance		:REAL;
	(* message if the assertion is false *)
	message			:AssertMessage;
END_VAR
IF (
	THIS^.isValueNaN(currentValue)
	OR_ELSE THIS^.isValueNaN(unexpectedValue)
	OR_ELSE THIS^.isValueNaN(tolerance)
) THEN
	RETURN;
ELSIF (THIS^.isValueInfinite(tolerance)) THEN
	THIS^.assertionWasWrong(message, THIS^.getDebugInfo('valueIsNotEqualTo'));
ELSIF (
	THIS^.isValueInfinite(currentValue)
	OR_ELSE THIS^.isValueInfinite(unexpectedValue)
) THEN
	RETURN (THIS^.isValuePositiveInfinite(currentValue) AND_THEN (NOT THIS^.isValuePositiveInfinite(unexpectedValue)));
	RETURN (THIS^.isValueNegativeInfinite(currentValue) AND_THEN (NOT THIS^.isValueNegativeInfinite(unexpectedValue)));
	RETURN (THIS^.isValuePositiveInfinite(unexpectedValue) AND_THEN (NOT THIS^.isValuePositiveInfinite(currentValue)));
	RETURN (THIS^.isValueNegativeInfinite(unexpectedValue) AND_THEN (NOT THIS^.isValueNegativeInfinite(currentValue)));
	THIS^.assertionWasWrong(message, THIS^.getDebugInfo('valueIsNotEqualTo'));
ELSIF (ABS(currentValue-unexpectedValue) <= ABS(tolerance)) THEN
	THIS^.assertionWasWrong(message, THIS^.getDebugInfo('valueIsNotEqualTo'));
END_IF
END_METHOD

(*

## Short summary
This assertion method checks if the current value is not negative infinite
NOT (-infinity), for details check [IEEE 754](https://en.wikipedia.org/wiki/IEEE_754)


.. <legal notes>

legal notes
=================
| SPDX-FileCopyrightText: © 2023 ekvip automation GmbH <info@ekvip.de>
| SPDX-License-Identifier: Apache-2.0
| For details check: Apache-2.0_

.. _Apache-2.0: https://www.apache.org/licenses/LICENSE-2.0

.. </legal notes>



*)

METHOD valueIsNotNegativeInfinite
VAR_INPUT
	(* current value to check *)
	currentValue	:REAL;
	(* message if the assertion is false *)
	message			:AssertMessage;
END_VAR
IF (THIS^.isValueNegativeInfinite(currentValue)) THEN
	THIS^.assertionWasWrong(message, THIS^.getDebugInfo('valueIsNotNegativeInfinite'));
END_IF
END_METHOD

(*

## Short summary
This assertion method checks if the current value is not positive infinite
NOT (infinity), for details check [IEEE 754](https://en.wikipedia.org/wiki/IEEE_754)


.. <legal notes>

legal notes
=================
| SPDX-FileCopyrightText: © 2023 ekvip automation GmbH <info@ekvip.de>
| SPDX-License-Identifier: Apache-2.0
| For details check: Apache-2.0_

.. _Apache-2.0: https://www.apache.org/licenses/LICENSE-2.0

.. </legal notes>



*)

METHOD valueIsNotPositiveInfinite
VAR_INPUT
	(* current value to check *)
	currentValue	:REAL;
	(* message if the assertion is false *)
	message			:AssertMessage;
END_VAR
IF (THIS^.isValuePositiveInfinite(currentValue)) THEN
	THIS^.assertionWasWrong(message, THIS^.getDebugInfo('valueIsNotPositiveInfinite'));
END_IF
END_METHOD

(*

## Short summary
This assertion method checks if the current value is a non special number
(NOT (NaN OR infinity OR -inifinity)), for details check [IEEE 754](https://en.wikipedia.org/wiki/IEEE_754)


.. <legal notes>

legal notes
=================
| SPDX-FileCopyrightText: © 2023 ekvip automation GmbH <info@ekvip.de>
| SPDX-License-Identifier: Apache-2.0
| For details check: Apache-2.0_

.. _Apache-2.0: https://www.apache.org/licenses/LICENSE-2.0

.. </legal notes>



*)

METHOD valueIsNotSpecial
VAR_INPUT
	(* current value to check *)
	currentValue	:REAL;
	(* message if the assertion is false *)
	message			:AssertMessage;
END_VAR
IF (THIS^.isValueSpecial(currentValue)) THEN
	THIS^.assertionWasWrong(message, THIS^.getDebugInfo('valueIsNotSpecial'));
END_IF
END_METHOD

(*

## Short summary
This assertion method checks if the current value is positve

**Attention:**
	Any comparsion to NaN is ``FALSE`` that means if ``currentValue``
	is NaN then is the assertion false.
	For details check `IEEE 754`_.

**Attention:**
	``currentValue`` has the value infinity means the assertion is true.
	``currentValue`` has the value -infinity means the assertion is false.
	``currentValue`` has the +0.0 means the assertion is true.
	``currentValue`` has the value -0.0 means the assertion is false.	
		For details check [IEEE 754](https://en.wikipedia.org/wiki/IEEE_754).


.. <legal notes>

legal notes
=================
| SPDX-FileCopyrightText: © 2022 ekvip automation GmbH <info@ekvip.de>
| SPDX-License-Identifier: Apache-2.0
| For details check: Apache-2.0_

.. _Apache-2.0: https://www.apache.org/licenses/LICENSE-2.0

.. </legal notes>



*)

METHOD valueIsPositive
VAR_INPUT
	(* current value to check *)
	currentValue	:REAL;
	(* message if the assertion is false *)
	message			:AssertMessage;
END_VAR
VAR
	(* just to cast ``currentValue`` *)
	currentValueAsDWord	:POINTER TO DWORD;
END_VAR
IF (THIS^.isValueNaN(currentValue)) THEN	
	THIS^.assertionWasWrong(message, THIS^.getDebugInfo('valueIsPositive'));
ELSE
	currentValueAsDWord := ADR(currentValue);
	IF ((currentValueAsDWord^ AND THIS^.MASK_FOR_SIGN_BIT) = THIS^.MASK_FOR_SIGN_BIT) THEN
		THIS^.assertionWasWrong(message, THIS^.getDebugInfo('valueIsPositive'));
	END_IF
END_IF
END_METHOD

(*

## Short summary
This assertion method checks if the current value is positive infinite
(infinity), for details check [IEEE 754](https://en.wikipedia.org/wiki/IEEE_754)


.. <legal notes>

legal notes
=================
| SPDX-FileCopyrightText: © 2023 ekvip automation GmbH <info@ekvip.de>
| SPDX-License-Identifier: Apache-2.0
| For details check: Apache-2.0_

.. _Apache-2.0: https://www.apache.org/licenses/LICENSE-2.0

.. </legal notes>



*)

METHOD valueIsPositiveInfinite
VAR_INPUT
	(* current value to check *)
	currentValue	:REAL;
	(* message if the assertion is false *)
	message			:AssertMessage;
END_VAR
IF (NOT THIS^.isValuePositiveInfinite(currentValue)) THEN
	THIS^.assertionWasWrong(message, THIS^.getDebugInfo('valueIsPositiveInfinite'));
END_IF
END_METHOD

(*

## Short summary
This assertion method checks if the current value is +0.0
for details check [IEEE 754](https://en.wikipedia.org/wiki/IEEE_754)


.. <legal notes>

legal notes
=================
| SPDX-FileCopyrightText: © 2023 ekvip automation GmbH <info@ekvip.de>
| SPDX-License-Identifier: Apache-2.0
| For details check: Apache-2.0_

.. _Apache-2.0: https://www.apache.org/licenses/LICENSE-2.0

.. </legal notes>



*)

METHOD valueIsPositiveZero
VAR_INPUT
	(* current value to check *)
	currentValue	:REAL;
	(* message if the assertion is false *)
	message			:AssertMessage;
END_VAR
VAR
	(* just to cast ``currentValue`` *)
	currentValueAsDWord	:POINTER TO DWORD;
END_VAR
currentValueAsDWord := ADR(currentValue);
IF (currentValueAsDWord^ <> THIS^.ZERO) THEN
	THIS^.assertionWasWrong(message, THIS^.getDebugInfo('valueIsPositiveZero'));
END_IF
END_METHOD

(*

## Short summary
This assertion method checks if the current value is a special
(NaN OR infinity OR -inifinity), for details check [IEEE 754](https://en.wikipedia.org/wiki/IEEE_754)


.. <legal notes>

legal notes
=================
| SPDX-FileCopyrightText: © 2023 ekvip automation GmbH <info@ekvip.de>
| SPDX-License-Identifier: Apache-2.0
| For details check: Apache-2.0_

.. _Apache-2.0: https://www.apache.org/licenses/LICENSE-2.0

.. </legal notes>



*)

METHOD valueIsSpecial
VAR_INPUT
	(* current value to check *)
	currentValue	:REAL;
	(* message if the assertion is false *)
	message			:AssertMessage;
END_VAR
IF (NOT THIS^.isValueSpecial(currentValue)) THEN
	THIS^.assertionWasWrong(message, THIS^.getDebugInfo('valueIsSpecial'));
END_IF
END_METHOD

(*

## Short summary
This assertion method checks if the current value is a subnormal number
for details check [IEEE 754](https://en.wikipedia.org/wiki/IEEE_754)


.. <legal notes>

legal notes
=================
| SPDX-FileCopyrightText: © 2023 ekvip automation GmbH <info@ekvip.de>
| SPDX-License-Identifier: Apache-2.0
| For details check: Apache-2.0_

.. _Apache-2.0: https://www.apache.org/licenses/LICENSE-2.0

.. </legal notes>



*)

METHOD valueIsSubnormal
VAR_INPUT
	(* current value to check *)
	currentValue	:REAL;
	(* message if the assertion is false *)
	message			:AssertMessage;
END_VAR
VAR
	(* just to cast ``currentValue`` *)
	currentValueAsDWord	:POINTER TO DWORD;
END_VAR
IF (THIS^.isValueNaN(currentValue)) THEN
	THIS^.assertionWasWrong(message, THIS^.getDebugInfo('valueIsSubnormal'));
ELSE
	currentValueAsDWord := ADR(currentValue);
	IF ((currentValueAsDWord^ AND THIS^.MASK_FOR_EXPONENT) <> THIS^.ZERO) THEN
		THIS^.assertionWasWrong(message, THIS^.getDebugInfo('valueIsSubnormal'));
	END_IF
END_IF
END_METHOD

END_FUNCTION_BLOCK

// ---- Assertor/Assertions/FloatAssertions/Lreal/classes/LrealAssertions.TcPOU
(*

## Short summary
This class provides assert statements for 64 bit floatings (``LREAL``).

.. <legal notes>

legal notes
=================
| SPDX-FileCopyrightText: © 2022 ekvip automation GmbH <info@ekvip.de>
| SPDX-License-Identifier: Apache-2.0
| For details check: Apache-2.0_

.. _Apache-2.0: https://www.apache.org/licenses/LICENSE-2.0

.. </legal notes>

*)

{attribute 'reflection'}
FUNCTION_BLOCK INTERNAL LrealAssertions EXTENDS AbstractAssertion IMPLEMENTS ILRealAssertions
VAR
END_VAR
VAR CONSTANT
	(* mask for determining value as a special value *)
	MASK_FOR_EXPONENT 	:LWORD := 16#7FF0_0000_0000_0000;
	(* mask for determining a special value as NaN or infinite *)  
	MASK_FOR_FRACTION	:LWORD := 16#000F_FFFF_FFFF_FFFF;
	(* mask to get the sign bit of an infinite or zero value *)
	MASK_FOR_SIGN_BIT	:LWORD := 16#8000_0000_0000_0000;
	(* just to compare results or the memory of a float value *)
	ZERO				:DWORD := 16#0000_0000_0000_0000;
END_VAR

(*

## Short summary
This abstract property returns the class name of the concrete object, 
It's for debugging purpose

.. <legal notes>

legal notes
=================
| SPDX-FileCopyrightText: © 2022 ekvip automation GmbH <info@ekvip.de>
| SPDX-License-Identifier: Apache-2.0
| For details check: Apache-2.0_

.. _Apache-2.0: https://www.apache.org/licenses/LICENSE-2.0

.. </legal notes>

*)

PROPERTY className :CNM_AbstractObject.ClassName
GET
className := 'CNM_Assertor.LrealAssertions';
END_GET
END_PROPERTY

(*

## Short summary
This method checks if a value is infinite
(infinity OR -inifinity), for details check [IEEE 754](https://en.wikipedia.org/wiki/IEEE_754)

.. <legal notes>

legal notes
=================
| SPDX-FileCopyrightText: © 2023 ekvip automation GmbH <info@ekvip.de>
| SPDX-License-Identifier: Apache-2.0
| For details check: Apache-2.0_

.. _Apache-2.0: https://www.apache.org/licenses/LICENSE-2.0

.. </legal notes>


:return: 
``TRUE``: value is inifinty or -infinity
``FALSE``: value is not inifinty and not -infinity

*)

METHOD PROTECTED isValueInfinite :BOOL
VAR_INPUT
	(* value to check *)
	value			:LREAL;	
END_VAR
VAR
	(* just to cast the value*)
	lrealAsLword	:POINTER TO LWORD;
END_VAR
lrealAsLword := ADR(value);
isValueInfinite := (
	THIS^.isValueSpecial(value)
	AND_THEN ((lrealAsLword^ AND THIS^.MASK_FOR_FRACTION) = THIS^.ZERO)
);
END_METHOD

(*

## Short summary
This method checks if a value is not a number
(NaN), for details check [IEEE 754](https://en.wikipedia.org/wiki/IEEE_754)

.. <legal notes>

legal notes
=================
| SPDX-FileCopyrightText: © 2023 ekvip automation GmbH <info@ekvip.de>
| SPDX-License-Identifier: Apache-2.0
| For details check: Apache-2.0_

.. _Apache-2.0: https://www.apache.org/licenses/LICENSE-2.0

.. </legal notes>


:return: 
``TRUE``: value is NaN
``FALSE``: value is not NaN

*)

METHOD PROTECTED isValueNaN :BOOL
VAR_INPUT
	(* value to check *)
	value			:LREAL;	
END_VAR
VAR
	(* just to cast the value*)
	lrealAsLword	:POINTER TO LWORD;
END_VAR
lrealAsLword := ADR(value);
isValueNaN := (
	THIS^.isValueSpecial(value)
	AND_THEN ((lrealAsLword^ AND THIS^.MASK_FOR_FRACTION) > THIS^.ZERO)
);
END_METHOD

(*

## Short summary
This method checks if a value is negative infinite
(-inifinity), for details check [IEEE 754](https://en.wikipedia.org/wiki/IEEE_754)


.. <legal notes>

legal notes
=================
| SPDX-FileCopyrightText: © 2023 ekvip automation GmbH <info@ekvip.de>
| SPDX-License-Identifier: Apache-2.0
| For details check: Apache-2.0_

.. _Apache-2.0: https://www.apache.org/licenses/LICENSE-2.0

.. </legal notes>


:return: 
``TRUE``: value is -infinity
``FALSE``: value is not -infinity

*)

{attribute 'analysis' := '-56'}
METHOD PROTECTED isValueNegativeInfinite : BOOL
VAR_INPUT
	(* value to check *)
	value			:LREAL;	
END_VAR
VAR
	(* just to cast the value*)
	lrealAsLword	:POINTER TO LWORD;
END_VAR
lrealAsLword := ADR(value);
isValueNegativeInfinite := (
	THIS^.isValueInfinite(value)
	AND_THEN ((lrealAsLword^ AND THIS^.MASK_FOR_SIGN_BIT) = THIS^.MASK_FOR_SIGN_BIT)
);
END_METHOD

(*

## Short summary
This method checks if a value is positive infinite
(infinity), for details check [IEEE 754](https://en.wikipedia.org/wiki/IEEE_754)


.. <legal notes>

legal notes
=================
| SPDX-FileCopyrightText: © 2023 ekvip automation GmbH <info@ekvip.de>
| SPDX-License-Identifier: Apache-2.0
| For details check: Apache-2.0_

.. _Apache-2.0: https://www.apache.org/licenses/LICENSE-2.0

.. </legal notes>


:return: 
``TRUE``: value is inifinty
``FALSE``: value is not inifinty

*)

METHOD PROTECTED isValuePositiveInfinite :BOOL
VAR_INPUT
	(* value to check *)
	value			:LREAL;	
END_VAR
VAR
	(* just to cast the value*)
	lrealAsLword	:POINTER TO LWORD;
END_VAR
lrealAsLword := ADR(value);
isValuePositiveInfinite := (
	THIS^.isValueInfinite(value)
	AND_THEN ((lrealAsLword^ AND THIS^.MASK_FOR_SIGN_BIT) = THIS^.ZERO)
);
END_METHOD

(*

## Short summary
This method checks if a value is a special value
(NaN OR infinity OR -inifinity), for details check [IEEE 754](https://en.wikipedia.org/wiki/IEEE_754)


.. <legal notes>

legal notes
=================
| SPDX-FileCopyrightText: © 2023 ekvip automation GmbH <info@ekvip.de>
| SPDX-License-Identifier: Apache-2.0
| For details check: Apache-2.0_

.. _Apache-2.0: https://www.apache.org/licenses/LICENSE-2.0

.. </legal notes>


:return: 
``TRUE``: value is inifinty or -infinity or NaN
``FALSE``: value is not inifinty and not -infinity and not NaN

*)

METHOD PROTECTED isValueSpecial :BOOL
VAR_INPUT
	(* value to check *)
	value			:LREAL;	
END_VAR
VAR
	(* just to cast the value*)
	lrealAsLword	:POINTER TO LWORD;
END_VAR
lrealAsLword := ADR(value);
isValueSpecial := ((lrealAsLword^ AND THIS^.MASK_FOR_EXPONENT) = THIS^.MASK_FOR_EXPONENT);
END_METHOD

(*

## Short summary
This assertion method checks if the current value is a number (NOT NaN)
for details check [IEEE 754](https://en.wikipedia.org/wiki/IEEE_754)


.. <legal notes>

legal notes
=================
| SPDX-FileCopyrightText: © 2023 ekvip automation GmbH <info@ekvip.de>
| SPDX-License-Identifier: Apache-2.0
| For details check: Apache-2.0_

.. _Apache-2.0: https://www.apache.org/licenses/LICENSE-2.0

.. </legal notes>



*)

METHOD valueIsANumber
VAR_INPUT
	(* current value to check *)
	currentValue	:LREAL;
	(* message if the assertion is false *)
	message			:AssertMessage;
END_VAR
IF (THIS^.isValueNaN(currentValue)) THEN
	THIS^.assertionWasWrong(message, THIS^.getDebugInfo('valueIsANumber'));
END_IF
END_METHOD

(*

## Short summary
This assertion method checks if the current value is equal to the expected value

**Attention:** 
	Nothing is equal to NaN, that means if ``currentValue`` OR ``expectedValue`` OR ``tolerance``
	is NaN then is the assertion false. For details check `IEEE 754`_

**Attention:** 
	infinity is equal to infinity and -infinity is equal to -infinity, that means if
	``currentValue`` AND ``expectedValue`` have the value infinity 
	OR ``currentValue`` AND ``expectedValue`` have the value -infinity
	the assertion is TRUE. For details check `IEEE 754`_

**Attention:** 
	If ``tolerance`` has the value infinity or -infinity and 
	``currentValue`` is not NaN and ``expectedValue`` is not NaN
	then is the assertion true. for details check [IEEE 754](https://en.wikipedia.org/wiki/IEEE_754)


.. <legal notes>

legal notes
=================
| SPDX-FileCopyrightText: © 2022 ekvip automation GmbH <info@ekvip.de>
| SPDX-License-Identifier: Apache-2.0
| For details check: Apache-2.0_

.. _Apache-2.0: https://www.apache.org/licenses/LICENSE-2.0

.. </legal notes>



*)

METHOD valueIsEqualTo
VAR_INPUT
	(* current value to check *)
	currentValue	:LREAL;
	(* expected value to compare *)
	expectedValue	:LREAL;
	(* tolerance to compensate twiddling floats, it has no sign *)
	tolerance		:LREAL;
	(* message if the assertion is false *)
	message			:AssertMessage;
END_VAR
IF (
	THIS^.isValueNaN(currentValue)
	OR_ELSE THIS^.isValueNaN(expectedValue)
	OR_ELSE THIS^.isValueNaN(tolerance)
) THEN
	THIS^.assertionWasWrong(message, THIS^.getDebugInfo('valueIsEqualTo'));
ELSIF (THIS^.isValueInfinite(tolerance)) THEN
	RETURN;
ELSIF (
	THIS^.isValueInfinite(currentValue)
	OR_ELSE THIS^.isValueInfinite(expectedValue)
	OR_ELSE THIS^.isValueInfinite(tolerance)
) THEN
	RETURN (THIS^.isValuePositiveInfinite(currentValue) AND_THEN THIS^.isValuePositiveInfinite(expectedValue));
	RETURN (THIS^.isValueNegativeInfinite(currentValue) AND_THEN THIS^.isValueNegativeInfinite(expectedValue));
	THIS^.assertionWasWrong(message, THIS^.getDebugInfo('valueIsEqualTo'));	
ELSIF (ABS(currentValue-expectedValue) > ABS(tolerance)) THEN
	THIS^.assertionWasWrong(message, THIS^.getDebugInfo('valueIsEqualTo'));
END_IF
END_METHOD

(*

## Short summary
This assertion method checks if the current value is finite
(NOT (infinity OR -inifinity)), for details check [IEEE 754](https://en.wikipedia.org/wiki/IEEE_754)


.. <legal notes>

legal notes
=================
| SPDX-FileCopyrightText: © 2023 ekvip automation GmbH <info@ekvip.de>
| SPDX-License-Identifier: Apache-2.0
| For details check: Apache-2.0_

.. _Apache-2.0: https://www.apache.org/licenses/LICENSE-2.0

.. </legal notes>



*)

METHOD valueIsFinite
VAR_INPUT
	(* current value to check *)
	currentValue	:LREAL;
	(* message if the assertion is false *)
	message			:AssertMessage;
END_VAR
IF (THIS^.isValueInfinite(currentValue)) THEN
	THIS^.assertionWasWrong(message, THIS^.getDebugInfo('valueIsFinite'));
END_IF
END_METHOD

(*

## Short summary
This assertion method checks if the current value is greater than the less value

**Attention:** 
	Any comparsion to NaN is ``FALSE`` that means if ``currentValue`` OR ``lessValue``
	is NaN then is the assertion false.
	For details check `IEEE 754`_ and the truth table below.

**Attention:** 
	Every number is smaller than infinity except infinity, it's equal.
	Every number is greater than -infinity except -infinity, it's equal.
	For details check [IEEE 754](https://en.wikipedia.org/wiki/IEEE_754) and the truth table below.


truth table for special values
===============================
+----------------------+-------------------+---------------+
| **``currentValue``** | **``lessValue``** | **assertion** |
+======================+===================+===============+
| NaN                  | Any value         | FASLE         |
+----------------------+-------------------+---------------+
| Any value            | NaN               | FALSE         |
+----------------------+-------------------+---------------+
| infinity             | NOT NaN           | TRUE          |
|                      | NOT infinity      |               |
+----------------------+-------------------+---------------+
| -infinity             | Any value         | FALSE         |
+----------------------+-------------------+---------------+
| Any value            | infinity          | FALSE         |
+----------------------+-------------------+---------------+
| NOT NaN              | -inifinity        | TRUE          |
| NOT -infinity        |                   |               |
+----------------------+-------------------+---------------+

.. <legal notes>

legal notes
=================
| SPDX-FileCopyrightText: © 2022 ekvip automation GmbH <info@ekvip.de>
| SPDX-License-Identifier: Apache-2.0
| For details check: Apache-2.0_

.. _Apache-2.0: https://www.apache.org/licenses/LICENSE-2.0

.. </legal notes>



*)

METHOD valueIsGreaterThan
VAR_INPUT
	(* current value to check *)
	currentValue	:LREAL;
	(* less than lower limit *)
	lessValue		:LREAL;
	(* message if the assertion is false *)
	message			:AssertMessage;
END_VAR
IF (
	THIS^.isValueNaN(currentValue) 
	OR_ELSE THIS^.isValueNaN(lessValue)
	OR_ELSE THIS^.isValueNegativeInfinite(currentValue) 
	OR_ELSE THIS^.isValuePositiveInfinite(lessValue)
)THEN
	THIS^.assertionWasWrong(message, THIS^.getDebugInfo('valueIsGreaterThan'));
ELSIF (
	THIS^.isValueNegativeInfinite(lessValue)
	OR_ELSE THIS^.isValuePositiveInfinite(currentValue)
) THEN
	RETURN;
ELSIF (currentValue <= lessValue) THEN
	THIS^.assertionWasWrong(message, THIS^.getDebugInfo('valueIsGreaterThan'));
END_IF
END_METHOD

(*

## Short summary
This assertion method checks if the current value is infinite
(infinity OR -inifinity), for details check [IEEE 754](https://en.wikipedia.org/wiki/IEEE_754)


.. <legal notes>

legal notes
=================
| SPDX-FileCopyrightText: © 2023 ekvip automation GmbH <info@ekvip.de>
| SPDX-License-Identifier: Apache-2.0
| For details check: Apache-2.0_

.. _Apache-2.0: https://www.apache.org/licenses/LICENSE-2.0

.. </legal notes>



*)

METHOD valueIsInfinite
VAR_INPUT
	(* current value to check *)
	currentValue	:LREAL;
	(* message if the assertion is false *)
	message			:AssertMessage;
END_VAR
IF (NOT THIS^.isValueInfinite(currentValue)) THEN
	THIS^.assertionWasWrong(message, THIS^.getDebugInfo('valueIsInfinite'));
END_IF
END_METHOD

(*

## Short summary
This assertion method checks if the current value is inside a limit

**Attention:** 
	limits are included: ``valueIsInRangeOf(3.0, 3.0, 3.0)`` is a true assertion

**Attention:** 
	Any comparsion to NaN is ``FALSE`` that means 
	if ``lowerLimit`` OR ``currentValue`` OR ``upperLimit``
	is NaN then is the assertion false.
	For details check `IEEE 754`_ and the truth table below.

**Attention:** 
	Every number is smaller than infinity except infinity, it's equal.
	Every number is greater than -infinity except -infinity, it's equal.
	For details check [IEEE 754](https://en.wikipedia.org/wiki/IEEE_754) and the truth table below.


truth table for special values
===============================
+--------------------+----------------------+--------------------+---------------+
| **``lowerLimit``** | **``currentValue``** | **``upperLimit``** | **assertion** |
+====================+======================+====================+===============+
| NaN                | Any value            | Any value          | FASLE         |
+--------------------+----------------------+--------------------+---------------+
| Any value          | NaN                  | Any value          | FALSE         |
+--------------------+----------------------+--------------------+---------------+
| Any value          | Any value            | NaN                | FALSE         |
+--------------------+----------------------+--------------------+---------------+
| -infinity          | NOT NaN              | infinity           | TRUE          |
+--------------------+----------------------+--------------------+---------------+
| infinity           | Any value            | -infinity          | FALSE         |
+--------------------+----------------------+--------------------+---------------+
| NOT -infinity      | -infinity            | Any value          | FALSE         |
+--------------------+----------------------+--------------------+---------------+
| Any value          | infinity             | NOT infinity       | FALSE         |
+--------------------+----------------------+--------------------+---------------+
| -infinity          | -infinity            | -infinity          | TRUE          |
+--------------------+----------------------+--------------------+---------------+
| infinity           | infinity             | infinity           | TRUE          |
+--------------------+----------------------+--------------------+---------------+
| -infinity          | NOT -infinity        | -infinity          | FALSE         |
+--------------------+----------------------+--------------------+---------------+
| infinity           | NOT infinity         | infinity           | FALSE         |
+--------------------+----------------------+--------------------+---------------+

.. <legal notes>

legal notes
=================
| SPDX-FileCopyrightText: © 2022 ekvip automation GmbH <info@ekvip.de>
| SPDX-License-Identifier: Apache-2.0
| For details check: Apache-2.0_

.. _Apache-2.0: https://www.apache.org/licenses/LICENSE-2.0

.. </legal notes>



*)

METHOD valueIsInRangeOf
VAR_INPUT
	(* lower limit for the current value *)
	lowerLimit		:LREAL;
	(* current value to check *)
	currentValue	:LREAL;
	(* upper limit for the current value *)
	upperLimit		:LREAL;
	(* message if the assertion is false *)
	message			:AssertMessage;
END_VAR
IF (
	THIS^.isValueNaN(lowerLimit)
	OR_ELSE THIS^.isValueNaN(currentValue)
	OR_ELSE THIS^.isValueNaN(upperLimit)
	OR_ELSE (
		THIS^.isValueNegativeInfinite(upperLimit) 
		AND_THEN THIS^.isValuePositiveInfinite(lowerLimit)
	) OR_ELSE (	
		THIS^.isValueNegativeInfinite(currentValue) 
		AND_THEN (NOT THIS^.isValueNegativeInfinite(lowerLimit))
	) OR_ELSE (
		THIS^.isValuePositiveInfinite(currentValue) 
		AND_THEN (NOT THIS^.isValuePositiveInfinite(upperLimit))
	) OR_ELSE (
		THIS^.isValuePositiveInfinite(lowerLimit)
		AND_THEN (NOT THIS^.isValuePositiveInfinite(currentValue))
		AND_THEN THIS^.isValuePositiveInfinite(upperLimit)
	) OR_ELSE (
		THIS^.isValueNegativeInfinite(lowerLimit)
		AND_THEN (NOT THIS^.isValueNegativeInfinite(currentValue))
		AND_THEN THIS^.isValueNegativeInfinite(upperLimit))
) THEN
	THIS^.assertionWasWrong(message, THIS^.getDebugInfo('valueIsInRangeOf'));
ELSIF ((
		THIS^.isValuePositiveInfinite(lowerLimit)
		AND_THEN THIS^.isValuePositiveInfinite(currentValue)
		AND_THEN THIS^.isValuePositiveInfinite(upperLimit)
	) OR_ELSE (
		THIS^.isValueNegativeInfinite(lowerLimit)
		AND_THEN THIS^.isValueNegativeInfinite(currentValue)
		AND_THEN THIS^.isValueNegativeInfinite(upperLimit)
	) OR_ELSE (
		THIS^.isValueNegativeInfinite(lowerLimit) 
		AND_THEN THIS^.isValuePositiveInfinite(upperLimit))
) THEN
	RETURN;
ELSIF ((currentValue < lowerLimit) OR (currentValue > upperLimit)) THEN
	THIS^.assertionWasWrong(message, THIS^.getDebugInfo('valueIsInRangeOf'));
END_IF
END_METHOD

(*

## Short summary
This assertion method checks if the current value is greater than the less value

**Attention:**
	Any comparsion to NaN is ``FALSE`` that means if ``currentValue`` OR ``greaterValue``
	is NaN then is the assertion false.
	For details check `IEEE 754`_ and the truth table below.

**Attention:**
	Every number is smaller than infinity except infinity, it's equal.
	Every number is greater than -infinity except -infinity, it's equal.
	For details check [IEEE 754](https://en.wikipedia.org/wiki/IEEE_754) and the truth table below.


truth table for special values
===============================
+----------------------+----------------------+---------------+
| **``currentValue``** | **``greaterValue``** | **assertion** |
+======================+======================+===============+
| NaN                  | Any value            | FASLE         |
+----------------------+----------------------+---------------+
| Any value            | NaN                  | FALSE         |
+----------------------+----------------------+---------------+
| infinity             | Any value            | FALSE         |
+----------------------+----------------------+---------------+
| -infinity             | NOT NaN              | TRUE          |
|                      | NOT -infinity        |               |
+----------------------+----------------------+---------------+
| NOT NaN              | infinity             | TRUE          |
| NOT infinity         |                      |               |
+----------------------+----------------------+---------------+

.. <legal notes>

legal notes
=================
| SPDX-FileCopyrightText: © 2022 ekvip automation GmbH <info@ekvip.de>
| SPDX-License-Identifier: Apache-2.0
| For details check: Apache-2.0_

.. _Apache-2.0: https://www.apache.org/licenses/LICENSE-2.0

.. </legal notes>



*)

METHOD valueIsLessThan
VAR_INPUT
	(* current value to check *)
	currentValue	:LREAL;
	(* greater than upper limit *)
	greaterValue	:LREAL;
	(* message if the assertion is false *)
	message			:AssertMessage;
END_VAR
IF (
	THIS^.isValueNaN(currentValue) 
	OR_ELSE THIS^.isValueNaN(greaterValue)
	OR_ELSE THIS^.isValuePositiveInfinite(currentValue)
	OR_ELSE THIS^.isValueNegativeInfinite(greaterValue)
) THEN
	THIS^.assertionWasWrong(message, THIS^.getDebugInfo('valueIsLessThan'));
ELSIF (
	THIS^.isValuePositiveInfinite(greaterValue)
	OR_ELSE THIS^.isValueNegativeInfinite(currentValue)
) THEN
	RETURN;
ELSIF (currentValue >= greaterValue) THEN
	THIS^.assertionWasWrong(message, THIS^.getDebugInfo('valueIsLessThan'));
END_IF
END_METHOD

(*

## Short summary
This assertion method checks if the current value is less than or equal to the maximum value

**Attention:**
	Any comparsion to NaN is ``FALSE`` that means if ``currentValue`` OR ``maximumValue``
	is NaN then is the assertion false.
	For details check `IEEE 754`_ and the truth table below.

**Attention:**
	Every number is smaller than infinity except infinity, it's equal.
	Every number is greater than -infinity except -infinity, it's equal.
	For details check [IEEE 754](https://en.wikipedia.org/wiki/IEEE_754) and the truth table below.


truth table for special values
===============================
+----------------------+----------------------+---------------+
| **``currentValue``** | **``maximumValue``** | **assertion** |
+======================+======================+===============+
| NaN                  | Any value            | FASLE         |
+----------------------+----------------------+---------------+
| Any value            | NaN                  | FALSE         |
+----------------------+----------------------+---------------+
| NOT NaN              | infinity             | TRUE          |
+----------------------+----------------------+---------------+
| -infinity            | NOT NaN              | TRUE          |
+----------------------+----------------------+---------------+
| infinity             | NOT infinity         | FALSE         |
+----------------------+----------------------+---------------+
| NOT -infinity        | -infinity            | FALSE         |
+----------------------+----------------------+---------------+

.. <legal notes>

legal notes
=================
| SPDX-FileCopyrightText: © 2022 ekvip automation GmbH <info@ekvip.de>
| SPDX-License-Identifier: Apache-2.0
| For details check: Apache-2.0_

.. _Apache-2.0: https://www.apache.org/licenses/LICENSE-2.0

.. </legal notes>



*)

METHOD valueIsMax
VAR_INPUT
	(* current value to check *)
	currentValue	:LREAL;
	(* upper limit for the current value *)
	maximumValue	:LREAL;
	(* message if the assertion is false *)
	message			:AssertMessage;
END_VAR
IF (
	THIS^.isValueNaN(currentValue) 
	OR_ELSE THIS^.isValueNaN(maximumValue)
	OR_ELSE (
		THIS^.isValueNegativeInfinite(maximumValue)
		AND_THEN (NOT THIS^.isValueNegativeInfinite(currentValue))
	) OR_ELSE (
		THIS^.isValuePositiveInfinite(currentValue)
		AND_THEN (NOT THIS^.isValuePositiveInfinite(maximumValue))
	)
) THEN
	THIS^.assertionWasWrong(message, THIS^.getDebugInfo('valueIsMax'));
ELSIF (
	THIS^.isValuePositiveInfinite(maximumValue)
	OR_ELSE THIS^.isValueNegativeInfinite(currentValue)
) THEN
	RETURN;
ELSIF (currentValue > maximumValue) THEN
	THIS^.assertionWasWrong(message, THIS^.getDebugInfo('valueIsMax'));
END_IF
END_METHOD

(*

## Short summary
This assertion method checks if the current value is greater than or equal to the minimum value

**Attention:**
	Any comparsion to NaN is ``FALSE`` that means if ``currentValue`` OR ``minimumValue``
	is NaN then is the assertion false.
	For details check `IEEE 754`_ and the truth table below.

**Attention:**
	Every number is smaller than infinity except infinity, it's equal.
	Every number is greater than -infinity except -infinity, it's equal.
	For details check [IEEE 754](https://en.wikipedia.org/wiki/IEEE_754) and the truth table below.


truth table for special values
===============================
+----------------------+----------------------+---------------+
| **``currentValue``** | **``minimumValue``** | **assertion** |
+======================+======================+===============+
| NaN                  | Any value            | FASLE         |
+----------------------+----------------------+---------------+
| Any value            | NaN                  | FALSE         |
+----------------------+----------------------+---------------+
| infinity             | NOT NaN              | TRUE          |
+----------------------+----------------------+---------------+
| NOT NaN              | -infinity            | TRUE          |
+----------------------+----------------------+---------------+
| -infinity            | NOT -infinity        | FALSE         |
+----------------------+----------------------+---------------+
| NOT infinity         | infinity             | FALSE         |
+----------------------+----------------------+---------------+

.. <legal notes>

legal notes
=================
| SPDX-FileCopyrightText: © 2022 ekvip automation GmbH <info@ekvip.de>
| SPDX-License-Identifier: Apache-2.0
| For details check: Apache-2.0_

.. _Apache-2.0: https://www.apache.org/licenses/LICENSE-2.0

.. </legal notes>



*)

METHOD valueIsMin
VAR_INPUT
	(* current value to check *)
	currentValue	:LREAL;
	(* lower limit for the current value *)
	minimumValue	:LREAL;
	(* message if the assertion is false *)
	message			:AssertMessage;
END_VAR
IF (
	THIS^.isValueNaN(currentValue) 
	OR_ELSE THIS^.isValueNaN(minimumValue)
	OR_ELSE (
		THIS^.isValueNegativeInfinite(currentValue)
		AND_THEN (NOT THIS^.isValueNegativeInfinite(minimumValue))
	) OR_ELSE (
		THIS^.isValuePositiveInfinite(minimumValue)
		AND_THEN (NOT THIS^.isValuePositiveInfinite(currentValue))
	)
) THEN
	THIS^.assertionWasWrong(message, THIS^.getDebugInfo('valueIsMin'));
ELSIF (
	THIS^.isValuePositiveInfinite(currentValue)
	OR_ELSE THIS^.isValueNegativeInfinite(minimumValue)
) THEN
	RETURN;
ELSIF (currentValue < minimumValue) THEN
	THIS^.assertionWasWrong(message, THIS^.getDebugInfo('valueIsMin'));
END_IF
END_METHOD

(*

## Short summary
This assertion method checks if the current value is a not a number (NaN)
for details check [IEEE 754](https://en.wikipedia.org/wiki/IEEE_754)


.. <legal notes>

legal notes
=================
| SPDX-FileCopyrightText: © 2023 ekvip automation GmbH <info@ekvip.de>
| SPDX-License-Identifier: Apache-2.0
| For details check: Apache-2.0_

.. _Apache-2.0: https://www.apache.org/licenses/LICENSE-2.0

.. </legal notes>



*)

METHOD valueIsNaN
VAR_INPUT
	(* current value to check *)
	currentValue	:LREAL;
	(* message if the assertion is false *)
	message			:AssertMessage;
END_VAR
IF (NOT THIS^.isValueNaN(currentValue)) THEN
	THIS^.assertionWasWrong(message, THIS^.getDebugInfo('valueIsNaN'));
END_IF
END_METHOD

(*

## Short summary
This assertion method checks if the current value is negative

**Attention:**
	Any comparsion to NaN is ``FALSE`` that means if ``currentValue``
	is NaN then is the assertion false.
	For details check `IEEE 754`_.

**Attention:**
	``currentValue`` has the value infinity means the assertion is false.
	``currentValue`` has the value -infinity means the assertion is true.
	``currentValue`` has the +0.0 means the assertion is false.
	``currentValue`` has the value -0.0 means the assertion is true.	
		For details check [IEEE 754](https://en.wikipedia.org/wiki/IEEE_754).


.. <legal notes>

legal notes
=================
| SPDX-FileCopyrightText: © 2022 ekvip automation GmbH <info@ekvip.de>
| SPDX-License-Identifier: Apache-2.0
| For details check: Apache-2.0_

.. _Apache-2.0: https://www.apache.org/licenses/LICENSE-2.0

.. </legal notes>



*)

METHOD valueIsNegative
VAR_INPUT
	(* current value to check *)
	currentValue	:LREAL;
	(* message if the assertion is false *)
	message			:AssertMessage;
END_VAR
VAR
	(* just to cast ``currentValue`` *)
	currentValueAsDWord	:POINTER TO LWORD;
END_VAR
IF (THIS^.isValueNaN(currentValue)) THEN	
	THIS^.assertionWasWrong(message, THIS^.getDebugInfo('valueIsNegative'));
ELSE
	currentValueAsDWord := ADR(currentValue);
	IF ((currentValueAsDWord^ AND THIS^.MASK_FOR_SIGN_BIT) = THIS^.ZERO) THEN
		THIS^.assertionWasWrong(message, THIS^.getDebugInfo('valueIsNegative'));
	END_IF
END_IF
END_METHOD

(*

## Short summary
This assertion method checks if the current value is negative infinite
(-infinity), for details check [IEEE 754](https://en.wikipedia.org/wiki/IEEE_754)


.. <legal notes>

legal notes
=================
| SPDX-FileCopyrightText: © 2023 ekvip automation GmbH <info@ekvip.de>
| SPDX-License-Identifier: Apache-2.0
| For details check: Apache-2.0_

.. _Apache-2.0: https://www.apache.org/licenses/LICENSE-2.0

.. </legal notes>



*)

METHOD valueIsNegativeInfinite
VAR_INPUT
	(* current value to check *)
	currentValue	:LREAL;
	(* message if the assertion is false *)
	message			:AssertMessage;
END_VAR
IF (NOT THIS^.isValueNegativeInfinite(currentValue)) THEN
	THIS^.assertionWasWrong(message, THIS^.getDebugInfo('valueIsNegativeInfinite'));
END_IF
END_METHOD

(*

## Short summary
This assertion method checks if the current value is -0.0
for details check [IEEE 754](https://en.wikipedia.org/wiki/IEEE_754)


.. <legal notes>

legal notes
=================
| SPDX-FileCopyrightText: © 2023 ekvip automation GmbH <info@ekvip.de>
| SPDX-License-Identifier: Apache-2.0
| For details check: Apache-2.0_

.. _Apache-2.0: https://www.apache.org/licenses/LICENSE-2.0

.. </legal notes>



*)

{attribute 'analysis' := '-56'}
METHOD valueIsNegativeZero
VAR_INPUT
	(* current value to check *)
	currentValue	:LREAL;
	(* message if the assertion is false *)
	message			:AssertMessage;
END_VAR
VAR
	(* just to cast ``currentValue`` *)
	currentValueAsDWord	:POINTER TO LWORD;
END_VAR
currentValueAsDWord := ADR(currentValue);
IF (currentValueAsDWord^ <> THIS^.MASK_FOR_SIGN_BIT) THEN
	THIS^.assertionWasWrong(message, THIS^.getDebugInfo('valueIsNegativeZero'));
END_IF
END_METHOD

(*

## Short summary
This assertion method checks if the current value is a normal number
(a finite non-zero/non-subnormal floating-point number)
for details check [IEEE 754](https://en.wikipedia.org/wiki/IEEE_754)


.. <legal notes>

legal notes
=================
| SPDX-FileCopyrightText: © 2023 ekvip automation GmbH <info@ekvip.de>
| SPDX-License-Identifier: Apache-2.0
| For details check: Apache-2.0_

.. _Apache-2.0: https://www.apache.org/licenses/LICENSE-2.0

.. </legal notes>



*)

METHOD valueIsNormal
VAR_INPUT
	(* current value to check *)
	currentValue	:LREAL;
	(* message if the assertion is false *)
	message			:AssertMessage;
END_VAR
VAR
	(* just to cast ``currentValue`` *)
	currentValueAsDWord	:POINTER TO LWORD;
END_VAR
IF (THIS^.isValueNaN(currentValue) OR_ELSE THIS^.isValueInfinite(currentValue)) THEN
	THIS^.assertionWasWrong(message, THIS^.getDebugInfo('valueIsNormal'));
ELSE
	currentValueAsDWord := ADR(currentValue);
	IF ((currentValueAsDWord^ AND THIS^.MASK_FOR_EXPONENT) = THIS^.ZERO) THEN
		THIS^.assertionWasWrong(message, THIS^.getDebugInfo('valueIsNormal'));
	END_IF
END_IF
END_METHOD

(*

## Short summary
This assertion method checks if the current value is not equal to the unexpected value

**Attention:** 
	Nothing is equal to NaN, that means if ``currentValue`` OR ``unexpectedValue`` OR ``tolerance``
	is NaN then is the assertion true. For details check `IEEE 754`_

**Attention:** 
	infinity is equal to infinity and -infinity is equal to -infinity, that means if
	``currentValue`` AND ``unexpectedValue`` have the value infinity 
	OR ``currentValue`` AND ``unexpectedValue`` have the value -infinity
	the assertion is false. For details check `IEEE 754`_

**Attention:** 
	If ``tolerance`` has the value infinity or -infinity and 
	``currentValue`` is not NaN and ``unexpectedValue`` is not NaN
	then is the assertion false. for details check [IEEE 754](https://en.wikipedia.org/wiki/IEEE_754)


.. <legal notes>

legal notes
=================
| SPDX-FileCopyrightText: © 2022 ekvip automation GmbH <info@ekvip.de>
| SPDX-License-Identifier: Apache-2.0
| For details check: Apache-2.0_

.. _Apache-2.0: https://www.apache.org/licenses/LICENSE-2.0

.. </legal notes>



*)

METHOD valueIsNotEqualTo
VAR_INPUT
	(* current value to check *)
	currentValue	:LREAL;
	(* unexpected value to compare *)
	unexpectedValue	:LREAL;
	(* tolerance to compensate twiddling floats, it has no sign *)
	tolerance		:LREAL;
	(* message if the assertion is false *)
	message			:AssertMessage;
END_VAR
IF (
	THIS^.isValueNaN(currentValue)
	OR_ELSE THIS^.isValueNaN(unexpectedValue)
	OR_ELSE THIS^.isValueNaN(tolerance)
) THEN
	RETURN;
ELSIF (THIS^.isValueInfinite(tolerance)) THEN
	THIS^.assertionWasWrong(message, THIS^.getDebugInfo('valueIsNotEqualTo'));
ELSIF (
	THIS^.isValueInfinite(currentValue)
	OR_ELSE THIS^.isValueInfinite(unexpectedValue)
) THEN
	RETURN (THIS^.isValuePositiveInfinite(currentValue) AND_THEN (NOT THIS^.isValuePositiveInfinite(unexpectedValue)));
	RETURN (THIS^.isValueNegativeInfinite(currentValue) AND_THEN (NOT THIS^.isValueNegativeInfinite(unexpectedValue)));
	RETURN (THIS^.isValuePositiveInfinite(unexpectedValue) AND_THEN (NOT THIS^.isValuePositiveInfinite(currentValue)));
	RETURN (THIS^.isValueNegativeInfinite(unexpectedValue) AND_THEN (NOT THIS^.isValueNegativeInfinite(currentValue)));
	THIS^.assertionWasWrong(message, THIS^.getDebugInfo('valueIsNotEqualTo'));
ELSIF (ABS(currentValue-unexpectedValue) <= ABS(tolerance)) THEN
	THIS^.assertionWasWrong(message, THIS^.getDebugInfo('valueIsNotEqualTo'));
END_IF
END_METHOD

(*

## Short summary
This assertion method checks if the current value is not negative infinite
NOT (-infinity), for details check [IEEE 754](https://en.wikipedia.org/wiki/IEEE_754)


.. <legal notes>

legal notes
=================
| SPDX-FileCopyrightText: © 2023 ekvip automation GmbH <info@ekvip.de>
| SPDX-License-Identifier: Apache-2.0
| For details check: Apache-2.0_

.. _Apache-2.0: https://www.apache.org/licenses/LICENSE-2.0

.. </legal notes>



*)

METHOD valueIsNotNegativeInfinite
VAR_INPUT
	(* current value to check *)
	currentValue	:LREAL;
	(* message if the assertion is false *)
	message			:AssertMessage;
END_VAR
IF (THIS^.isValueNegativeInfinite(currentValue)) THEN
	THIS^.assertionWasWrong(message, THIS^.getDebugInfo('valueIsNotNegativeInfinite'));
END_IF
END_METHOD

(*

## Short summary
This assertion method checks if the current value is not positive infinite
NOT (infinity), for details check [IEEE 754](https://en.wikipedia.org/wiki/IEEE_754)


.. <legal notes>

legal notes
=================
| SPDX-FileCopyrightText: © 2023 ekvip automation GmbH <info@ekvip.de>
| SPDX-License-Identifier: Apache-2.0
| For details check: Apache-2.0_

.. _Apache-2.0: https://www.apache.org/licenses/LICENSE-2.0

.. </legal notes>



*)

METHOD valueIsNotPositiveInfinite
VAR_INPUT
	(* current value to check *)
	currentValue	:LREAL;
	(* message if the assertion is false *)
	message			:AssertMessage;
END_VAR
IF (THIS^.isValuePositiveInfinite(currentValue)) THEN
	THIS^.assertionWasWrong(message, THIS^.getDebugInfo('valueIsNotPositiveInfinite'));
END_IF
END_METHOD

(*

## Short summary
This assertion method checks if the current value is a non special number
(NOT (NaN OR infinity OR -inifinity)), for details check [IEEE 754](https://en.wikipedia.org/wiki/IEEE_754)


.. <legal notes>

legal notes
=================
| SPDX-FileCopyrightText: © 2023 ekvip automation GmbH <info@ekvip.de>
| SPDX-License-Identifier: Apache-2.0
| For details check: Apache-2.0_

.. _Apache-2.0: https://www.apache.org/licenses/LICENSE-2.0

.. </legal notes>



*)

METHOD valueIsNotSpecial
VAR_INPUT
	(* current value to check *)
	currentValue	:LREAL;
	(* message if the assertion is false *)
	message			:AssertMessage;
END_VAR
IF (THIS^.isValueSpecial(currentValue)) THEN
	THIS^.assertionWasWrong(message, THIS^.getDebugInfo('valueIsNotSpecial'));
END_IF
END_METHOD

(*

## Short summary
This assertion method checks if the current value is positve

**Attention:**
	Any comparsion to NaN is ``FALSE`` that means if ``currentValue``
	is NaN then is the assertion false.
	For details check `IEEE 754`_.

**Attention:**
	``currentValue`` has the value infinity means the assertion is true.
	``currentValue`` has the value -infinity means the assertion is false.
	``currentValue`` has the +0.0 means the assertion is true.
	``currentValue`` has the value -0.0 means the assertion is false.	
		For details check [IEEE 754](https://en.wikipedia.org/wiki/IEEE_754).


.. <legal notes>

legal notes
=================
| SPDX-FileCopyrightText: © 2022 ekvip automation GmbH <info@ekvip.de>
| SPDX-License-Identifier: Apache-2.0
| For details check: Apache-2.0_

.. _Apache-2.0: https://www.apache.org/licenses/LICENSE-2.0

.. </legal notes>



*)

{attribute 'analysis' := '-56'}
METHOD valueIsPositive
VAR_INPUT
	(* current value to check *)
	currentValue	:LREAL;
	(* message if the assertion is false *)
	message			:AssertMessage;
END_VAR
VAR
	(* just to cast ``currentValue`` *)
	currentValueAsDWord	:POINTER TO LWORD;
END_VAR
IF (THIS^.isValueNaN(currentValue)) THEN	
	THIS^.assertionWasWrong(message, THIS^.getDebugInfo('valueIsPositive'));
ELSE
	currentValueAsDWord := ADR(currentValue);
	IF ((currentValueAsDWord^ AND THIS^.MASK_FOR_SIGN_BIT) = THIS^.MASK_FOR_SIGN_BIT) THEN
		THIS^.assertionWasWrong(message, THIS^.getDebugInfo('valueIsPositive'));
	END_IF
END_IF
END_METHOD

(*

## Short summary
This assertion method checks if the current value is positive infinite
(infinity), for details check [IEEE 754](https://en.wikipedia.org/wiki/IEEE_754)


.. <legal notes>

legal notes
=================
| SPDX-FileCopyrightText: © 2023 ekvip automation GmbH <info@ekvip.de>
| SPDX-License-Identifier: Apache-2.0
| For details check: Apache-2.0_

.. _Apache-2.0: https://www.apache.org/licenses/LICENSE-2.0

.. </legal notes>



*)

METHOD valueIsPositiveInfinite
VAR_INPUT
	(* current value to check *)
	currentValue	:LREAL;
	(* message if the assertion is false *)
	message			:AssertMessage;
END_VAR
IF (NOT THIS^.isValuePositiveInfinite(currentValue)) THEN
	THIS^.assertionWasWrong(message, THIS^.getDebugInfo('valueIsPositiveInfinite'));
END_IF
END_METHOD

(*

## Short summary
This assertion method checks if the current value is +0.0
for details check [IEEE 754](https://en.wikipedia.org/wiki/IEEE_754)


.. <legal notes>

legal notes
=================
| SPDX-FileCopyrightText: © 2023 ekvip automation GmbH <info@ekvip.de>
| SPDX-License-Identifier: Apache-2.0
| For details check: Apache-2.0_

.. _Apache-2.0: https://www.apache.org/licenses/LICENSE-2.0

.. </legal notes>



*)

METHOD valueIsPositiveZero
VAR_INPUT
	(* current value to check *)
	currentValue	:LREAL;
	(* message if the assertion is false *)
	message			:AssertMessage;
END_VAR
VAR
	(* just to cast ``currentValue`` *)
	currentValueAsDWord	:POINTER TO LWORD;
END_VAR
currentValueAsDWord := ADR(currentValue);
IF (currentValueAsDWord^ <> THIS^.ZERO) THEN
	THIS^.assertionWasWrong(message, THIS^.getDebugInfo('valueIsPositiveZero'));
END_IF
END_METHOD

(*

## Short summary
This assertion method checks if the current value is a special
(NaN OR infinity OR -inifinity), for details check [IEEE 754](https://en.wikipedia.org/wiki/IEEE_754)


.. <legal notes>

legal notes
=================
| SPDX-FileCopyrightText: © 2023 ekvip automation GmbH <info@ekvip.de>
| SPDX-License-Identifier: Apache-2.0
| For details check: Apache-2.0_

.. _Apache-2.0: https://www.apache.org/licenses/LICENSE-2.0

.. </legal notes>



*)

METHOD valueIsSpecial
VAR_INPUT
	(* current value to check *)
	currentValue	:LREAL;
	(* message if the assertion is false *)
	message			:AssertMessage;
END_VAR
IF (NOT THIS^.isValueSpecial(currentValue)) THEN
	THIS^.assertionWasWrong(message, THIS^.getDebugInfo('valueIsSpecial'));
END_IF
END_METHOD

(*

## Short summary
This assertion method checks if the current value is a subnormal number
for details check [IEEE 754](https://en.wikipedia.org/wiki/IEEE_754)


.. <legal notes>

legal notes
=================
| SPDX-FileCopyrightText: © 2023 ekvip automation GmbH <info@ekvip.de>
| SPDX-License-Identifier: Apache-2.0
| For details check: Apache-2.0_

.. _Apache-2.0: https://www.apache.org/licenses/LICENSE-2.0

.. </legal notes>



*)

METHOD valueIsSubnormal
VAR_INPUT
	(* current value to check *)
	currentValue	:LREAL;
	(* message if the assertion is false *)
	message			:AssertMessage;
END_VAR
VAR
	(* just to cast ``currentValue`` *)
	currentValueAsDWord	:POINTER TO LWORD;
END_VAR
IF (THIS^.isValueNaN(currentValue)) THEN
	THIS^.assertionWasWrong(message, THIS^.getDebugInfo('valueIsSubnormal'));
ELSE
	currentValueAsDWord := ADR(currentValue);
	IF ((currentValueAsDWord^ AND THIS^.MASK_FOR_EXPONENT) <> THIS^.ZERO) THEN
		THIS^.assertionWasWrong(message, THIS^.getDebugInfo('valueIsSubnormal'));
	END_IF
END_IF
END_METHOD

END_FUNCTION_BLOCK

// ---- Assertor/Assertions/IntegerAssertions/classes/IntegerAssertions.TcPOU
(*

## Short summary

This class provides assert statements for signed/unsigned integers from 8~64 bit length.
For signed integers use `IntegerAssertions.signed`
For unsigned integers use `IntegerAssertions.unsigned`

.. <legal notes>

legal notes
=================
| SPDX-FileCopyrightText: © 2022 ekvip automation GmbH <info@ekvip.de>
| SPDX-License-Identifier: Apache-2.0
| For details check: Apache-2.0_

.. _Apache-2.0: https://www.apache.org/licenses/LICENSE-2.0

.. </legal notes>

methods aand properties
========================

*)

{attribute 'reflection'}
FUNCTION_BLOCK INTERNAL IntegerAssertions EXTENDS CNM_AbstractObject.Object IMPLEMENTS IIntegerAssertions, IAssertCallBacksetter
VAR
	(* class to handle assert statements for signed integers *)
	signedIntegerAssertions		:SignedIntegerAssertions();
	(* class to handle assert statements for unsigned integers *)
	unsignedIntegerAssertions	:UnsignedIntegerAssertions();
END_VAR

(*

## Short summary
This abstract property returns the class name of the concrete object, 
It's for debugging purpose

.. <legal notes>

legal notes
=================
| SPDX-FileCopyrightText: © 2022 ekvip automation GmbH <info@ekvip.de>
| SPDX-License-Identifier: Apache-2.0
| For details check: Apache-2.0_

.. _Apache-2.0: https://www.apache.org/licenses/LICENSE-2.0

.. </legal notes>

*)

PROPERTY className :CNM_AbstractObject.ClassName
GET
className := 'CNM_AssertionInterfaceLib.IntegerAssertions';
END_GET
END_PROPERTY

(*

## Short summary
This methods is the setter for the callback class if an assertion was false

.. <legal notes>

legal notes
=================
| SPDX-FileCopyrightText: © 2022 ekvip automation GmbH <info@ekvip.de>
| SPDX-License-Identifier: Apache-2.0
| For details check: Apache-2.0_

.. _Apache-2.0: https://www.apache.org/licenses/LICENSE-2.0

.. </legal notes>



*)

METHOD setCallBack
VAR_INPUT
	(* the class that must be informed if an assertion is false *)
	callBack	:IAssertCallBack;  
END_VAR
THIS^.signedIntegerAssertions.setCallBack(callBack);
THIS^.unsignedIntegerAssertions.setCallBack(callBack);
END_METHOD

(*

## Short summary
Returns the interface `ISignedIntegerAssertions` with assert statements for signed integers from 8~64 bit length 

.. <legal notes>

legal notes
=================
| SPDX-FileCopyrightText: © 2022 ekvip automation GmbH <info@ekvip.de>
| SPDX-License-Identifier: Apache-2.0
| For details check: Apache-2.0_

.. _Apache-2.0: https://www.apache.org/licenses/LICENSE-2.0

.. </legal notes>

*)

PROPERTY signed :ISignedIntegerAssertions
GET
signed := THIS^.signedIntegerAssertions;
END_GET
END_PROPERTY

(*

## Short summary
Returns the interface `IUnsignedIntegerAssertions` with assert statements for unsigned integers from 8~64 bit length 

.. <legal notes>

legal notes
=================
| SPDX-FileCopyrightText: © 2022 ekvip automation GmbH <info@ekvip.de>
| SPDX-License-Identifier: Apache-2.0
| For details check: Apache-2.0_

.. _Apache-2.0: https://www.apache.org/licenses/LICENSE-2.0

.. </legal notes>

*)

PROPERTY unsigned :IUnsignedIntegerAssertions
GET
unsigned := THIS^.unsignedIntegerAssertions;
END_GET
END_PROPERTY

END_FUNCTION_BLOCK

// ---- Assertor/Assertions/IntegerAssertions/signed/classes/SignedIntegerAssertions.TcPOU
(*

## Short summary

This class provides assert statements for signed integers from 8~64 bit length 
For 8 bit integers use `SignedIntegerAssertions.short`
For 16 bit integers use `SignedIntegerAssertions.simple`
For 32 bit integers use `SignedIntegerAssertions.double`
For 64 bit integers use `SignedIntegerAssertions.long`
For integers in register length use `SignedIntegerAssertions.x`

.. <legal notes>

legal notes
=================
| SPDX-FileCopyrightText: © 2022 ekvip automation GmbH <info@ekvip.de>
| SPDX-License-Identifier: Apache-2.0
| For details check: Apache-2.0_

.. _Apache-2.0: https://www.apache.org/licenses/LICENSE-2.0

.. </legal notes>



*)

{attribute 'reflection'}
FUNCTION_BLOCK INTERNAL SignedIntegerAssertions EXTENDS CNM_AbstractObject.Object IMPLEMENTS ISignedIntegerAssertions, IAssertCallBacksetter
VAR
	(* class to handle assert statements for signed short integers *)
	sintAssertions	:SintAssertions();
	(* class to handle assert statements for signed integers *)
	intAssertions	:IntAssertions();
	(* class to handle assert statements for signed double integers *)
	dintAssertions	:DintAssertions();
	(* class to handle assert statements for signed register length integers *)
	xintAssertions	:XintAssertions();
	(* class to handle assert statements for signed long integers *)
	lintAssertions	:LintAssertions();
END_VAR

(*

## Short summary
This abstract property returns the class name of the concrete object, 
It's for debugging purpose

.. <legal notes>

legal notes
=================
| SPDX-FileCopyrightText: © 2022 ekvip automation GmbH <info@ekvip.de>
| SPDX-License-Identifier: Apache-2.0
| For details check: Apache-2.0_

.. _Apache-2.0: https://www.apache.org/licenses/LICENSE-2.0

.. </legal notes>

*)

PROPERTY className :CNM_AbstractObject.ClassName
GET
className := 'CNM_Assertor.SignedIntegerAssertions';
END_GET
END_PROPERTY

(*

